C03634=1025.700,9.910,403.538,167.481,46.945,158.663
C03635=1025.707,10.159,403.524,167.485,46.942,158.663
C03636=1025.713,10.408,403.509,167.487,46.939,158.663
C03637=1025.719,10.658,403.495,167.489,46.937,158.663
C03638=1025.725,10.908,403.480,167.492,46.933,158.662
C03639=1025.731,11.192,403.463,167.495,46.930,158.662
C03640=1025.739,11.476,403.446,167.498,46.926,158.662
C03641=1025.745,11.760,403.429,167.501,46.922,158.661
C03642=1025.753,12.044,403.413,167.504,46.919,158.661
C03643=1025.759,12.293,403.398,167.506,46.916,158.661
C03644=1025.765,12.542,403.383,167.510,46.913,158.661
C03645=1025.772,12.792,403.368,167.512,46.910,158.660
C03646=1025.777,13.041,403.354,167.515,46.907,158.660
C03647=1025.784,13.291,403.339,167.517,46.903,158.660
C03648=1025.790,13.540,403.324,167.519,46.900,158.660
C03649=1025.797,13.790,403.309,167.522,46.897,158.659
C03650=1025.802,14.039,403.294,167.525,46.895,158.659
C03651=1025.809,14.289,403.279,167.528,46.892,158.659
C03652=1025.815,14.538,403.264,167.530,46.889,158.659
C03653=1025.821,14.788,403.249,167.532,46.886,158.659
C03654=1025.827,15.037,403.234,167.535,46.883,158.658
C03655=1025.833,15.287,403.219,167.538,46.880,158.658
C03656=1025.839,15.537,403.204,167.541,46.877,158.658
C03657=1025.845,15.785,403.188,167.543,46.874,158.658
C03658=1025.851,16.035,403.173,167.545,46.871,158.657
C03659=1025.857,16.285,403.158,167.548,46.868,158.657
C03660=1025.864,16.534,403.144,167.550,46.865,158.657
C03661=1025.870,16.783,403.129,167.554,46.862,158.657
C03662=1025.875,17.033,403.113,167.556,46.859,158.656
C03663=1025.882,17.283,403.098,167.558,46.856,158.656
C03664=1025.888,17.532,403.083,167.561,46.853,158.656
C03665=1025.895,17.781,403.068,167.563,46.850,158.656
C03666=1025.900,18.031,403.053,167.567,46.847,158.655
C03667=1025.906,18.280,403.038,167.569,46.844,158.655
C03668=1025.912,18.530,403.023,167.571,46.841,158.655
C03669=1025.919,18.780,403.008,167.574,46.838,158.655
C03670=1025.924,19.028,402.992,167.576,46.835,158.655
C03671=1025.931,19.278,402.977,167.580,46.832,158.654
C03672=1025.937,19.528,402.962,167.582,46.829,158.654
C03673=1025.943,19.777,402.947,167.584,46.826,158.654
C03674=1025.949,20.027,402.931,167.587,46.823,158.653
C03675=1025.956,20.276,402.916,167.589,46.820,158.653
C03676=1025.961,20.526,402.901,167.591,46.817,158.653
C03677=1025.967,20.775,402.885,167.595,46.814,158.653
C03678=1025.974,21.024,402.870,167.597,46.811,158.653
C03679=1025.979,21.274,402.855,167.599,46.808,158.652
C03680=1025.986,21.524,402.840,167.602,46.805,158.652
C03681=1025.991,21.773,402.824,167.605,46.803,158.652
C03682=1025.998,22.022,402.809,167.607,46.799,158.652
C03683=1026.004,22.272,402.794,167.610,46.796,158.651
C03684=1026.010,22.521,402.778,167.612,46.793,158.651
C03685=1026.016,22.771,402.763,167.615,46.790,158.651
C03686=1026.023,23.020,402.747,167.617,46.787,158.651
C03687=1026.029,23.270,402.731,167.620,46.785,158.650
C03688=1026.034,23.519,402.717,167.623,46.782,158.650
C03689=1026.040,23.768,402.701,167.625,46.779,158.650
C03690=1026.047,24.018,402.686,167.628,46.775,158.650
C03691=1026.053,24.267,402.671,167.630,46.772,158.649
C03692=1026.059,24.517,402.654,167.632,46.769,158.649
C03693=1026.065,24.766,402.639,167.636,46.766,158.649
C03694=1026.071,25.016,402.623,167.638,46.764,158.649
C03695=1026.078,25.266,402.608,167.640,46.761,158.648
C03696=1026.084,25.514,402.593,167.643,46.758,158.648
C03697=1026.090,25.764,402.577,167.645,46.754,158.648
C03698=1026.096,26.013,402.563,167.648,46.751,158.648
C03699=1026.102,26.263,402.546,167.651,46.748,158.647
C03700=1026.108,26.512,402.531,167.653,46.746,158.647
C03701=1026.114,26.762,402.515,167.656,46.743,158.647
C03702=1026.121,27.011,402.500,167.658,46.740,158.647
C03703=1026.127,27.297,402.482,167.661,46.736,158.646
C03704=1026.135,27.582,402.464,167.664,46.732,158.646
C03705=1026.142,27.867,402.446,167.668,46.729,158.646
C03706=1026.149,28.152,402.429,167.669,46.726,158.645
C03707=1026.154,28.402,402.413,167.673,46.723,158.645
C03708=1026.161,28.651,402.397,167.675,46.720,158.645
C03709=1026.167,28.901,402.382,167.677,46.717,158.645
C03710=1026.173,29.151,402.366,167.680,46.714,158.645
C03711=1026.179,29.400,402.350,167.683,46.711,158.644
C03712=1026.185,29.650,402.334,167.685,46.709,158.644
C03713=1026.191,29.899,402.318,167.688,46.706,158.644
C03714=1026.198,30.148,402.302,167.690,46.703,158.644
C03715=1026.203,30.398,402.287,167.692,46.700,158.643
C03716=1026.210,30.647,402.271,167.695,46.696,158.643
C03717=1026.216,30.896,402.255,167.698,46.693,158.643
C03718=1026.221,31.146,402.239,167.700,46.691,158.643
C03719=1026.228,31.395,402.224,167.703,46.688,158.642
C03720=1026.234,31.645,402.208,167.705,46.685,158.642
C03721=1026.240,31.895,402.192,167.708,46.682,158.642
C03722=1026.246,32.144,402.176,167.711,46.679,158.642
C03723=1026.252,32.393,402.160,167.713,46.676,158.641
C03724=1026.258,32.643,402.145,167.715,46.673,158.641
C03725=1026.265,32.892,402.129,167.718,46.670,158.641
C03726=1026.271,33.141,402.113,167.720,46.667,158.641
C03727=1026.276,33.391,402.097,167.723,46.664,158.640
C03728=1026.283,33.640,402.081,167.726,46.661,158.640
C03729=1026.289,33.890,402.065,167.728,46.658,158.640
C03730=1026.296,34.139,402.049,167.730,46.656,158.640
C03731=1026.301,34.389,402.034,167.734,46.652,158.639
C03732=1026.307,34.638,402.018,167.735,46.649,158.639
C03733=1026.314,34.887,402.002,167.738,46.646,158.639
C03734=1026.320,35.136,401.986,167.741,46.643,158.639
C03735=1026.326,35.386,401.970,167.743,46.640,158.638
C03736=1026.332,35.635,401.955,167.745,46.638,158.638
C03737=1026.338,35.885,401.938,167.749,46.635,158.638
C03738=1026.344,36.134,401.922,167.751,46.631,158.638
C03739=1026.351,36.383,401.906,167.753,46.628,158.637
C03740=1026.356,36.633,401.891,167.756,46.625,158.637
C03741=1026.362,36.883,401.875,167.758,46.623,158.637
C03742=1026.368,37.132,401.858,167.760,46.620,158.637
C03743=1026.375,37.381,401.843,167.764,46.617,158.636
C03744=1026.382,37.631,401.826,167.766,46.614,158.636
C03745=1026.388,37.880,401.810,167.768,46.611,158.636
C03746=1026.394,38.130,401.794,167.770,46.608,158.635
C03747=1026.399,38.379,401.777,167.773,46.605,158.635
C03748=1026.405,38.628,401.761,167.776,46.602,158.635
C03749=1026.411,38.878,401.745,167.778,46.599,158.635
C03750=1026.417,39.127,401.729,167.781,46.596,158.635
C03751=1026.423,39.376,401.712,167.783,46.593,158.634
C03752=1026.430,39.625,401.697,167.785,46.590,158.634
C03753=1026.436,39.875,401.680,167.789,46.587,158.634
C03754=1026.442,40.124,401.664,167.791,46.585,158.634
C03755=1026.448,40.373,401.648,167.793,46.582,158.633
C03756=1026.454,40.624,401.631,167.795,46.579,158.633
C03757=1026.460,40.873,401.615,167.798,46.575,158.633
C03758=1026.466,41.122,401.599,167.801,46.573,158.632
C03759=1026.472,41.372,401.582,167.803,46.570,158.632
C03760=1026.478,41.621,401.566,167.806,46.567,158.632
C03761=1026.484,41.870,401.550,167.808,46.564,158.632
C03762=1026.491,42.119,401.534,167.810,46.561,158.632
C03763=1026.497,42.369,401.518,167.814,46.558,158.631
C03764=1026.503,42.619,401.501,167.816,46.555,158.631
C03765=1026.509,42.868,401.485,167.818,46.553,158.631
C03766=1026.515,43.117,401.469,167.820,46.550,158.631
C03767=1026.522,43.403,401.449,167.823,46.546,158.630
C03768=1026.528,43.688,401.431,167.827,46.543,158.630
C03769=1026.535,43.973,401.412,167.829,46.540,158.630
C03770=1026.542,44.259,401.393,167.832,46.537,158.629
C03771=1026.548,44.508,401.377,167.834,46.534,158.629
C03772=1026.554,44.758,401.360,167.837,46.531,158.629
C03773=1026.560,45.007,401.343,167.839,46.528,158.629
C03774=1026.566,45.256,401.327,167.842,46.525,158.628
C03775=1026.571,45.506,401.310,167.844,46.523,158.628
C03776=1026.578,45.755,401.293,167.847,46.520,158.628
C03777=1026.584,46.004,401.277,167.849,46.517,158.628
C03778=1026.590,46.254,401.260,167.852,46.514,158.628
C03779=1026.596,46.504,401.244,167.854,46.511,158.627
C03780=1026.602,46.753,401.227,167.857,46.508,158.627
C03781=1026.608,47.002,401.210,167.859,46.505,158.627
C03782=1026.614,47.251,401.194,167.862,46.503,158.627
C03783=1026.620,47.501,401.177,167.864,46.500,158.626
C03784=1026.626,47.750,401.160,167.867,46.497,158.626
C03785=1026.632,48.000,401.144,167.869,46.494,158.626
C03786=1026.638,48.249,401.127,167.871,46.491,158.626
C03787=1026.644,48.498,401.110,167.874,46.489,158.625
C03788=1026.650,48.748,401.094,167.877,46.486,158.625
C03789=1026.656,48.997,401.077,167.879,46.482,158.625
C03790=1026.662,49.247,401.061,167.881,46.479,158.624
C03791=1026.668,49.496,401.044,167.883,46.477,158.624
C03792=1026.674,49.745,401.027,167.887,46.474,158.624
C03793=1026.680,49.995,401.011,167.889,46.471,158.624
C03794=1026.687,50.244,400.994,167.891,46.468,158.624
C03795=1026.693,50.493,400.978,167.893,46.465,158.623
C03796=1026.698,50.742,400.960,167.897,46.462,158.623
C03797=1026.705,50.992,400.943,167.899,46.460,158.623
C03798=1026.711,51.241,400.927,167.901,46.457,158.623
C03799=1026.717,51.490,400.910,167.904,46.454,158.622
C03800=1026.723,51.740,400.894,167.906,46.451,158.622
C03801=1026.729,51.990,400.877,167.908,46.448,158.622
C03802=1026.735,52.239,400.860,167.911,46.445,158.621
C03803=1026.741,52.488,400.843,167.914,46.442,158.621
C03804=1026.748,52.737,400.826,167.916,46.439,158.621
C03805=1026.753,52.987,400.809,167.918,46.436,158.621
C03806=1026.759,53.236,400.793,167.922,46.433,158.621
C03807=1026.765,53.485,400.776,167.924,46.430,158.620
C03808=1026.772,53.735,400.759,167.926,46.428,158.620
C03809=1026.778,53.984,400.742,167.928,46.424,158.620
C03810=1026.783,54.234,400.726,167.931,46.421,158.619
C03811=1026.790,54.483,400.708,167.933,46.418,158.619
C03812=1026.796,54.732,400.692,167.936,46.416,158.619
C03813=1026.802,54.981,400.675,167.939,46.413,158.619
C03814=1026.809,55.231,400.658,167.941,46.410,158.618
C03815=1026.814,55.480,400.641,167.943,46.407,158.618
C03816=1026.820,55.730,400.625,167.945,46.404,158.618
C03817=1026.827,55.979,400.607,167.949,46.401,158.618
C03818=1026.833,56.228,400.591,167.951,46.398,158.617
C03819=1026.838,56.477,400.573,167.953,46.395,158.617
C03820=1026.845,56.727,400.557,167.956,46.392,158.617
C03821=1026.851,56.976,400.540,167.958,46.389,158.616
C03822=1026.858,57.226,400.523,167.961,46.386,158.616
C03823=1026.863,57.475,400.506,167.963,46.383,158.616
C03824=1026.869,57.725,400.489,167.966,46.380,158.616
C03825=1026.876,57.974,400.472,167.968,46.377,158.615
C03826=1026.882,58.223,400.456,167.970,46.374,158.615
C03827=1026.888,58.472,400.439,167.973,46.371,158.615
C03828=1026.895,58.722,400.421,167.976,46.368,158.615
C03829=1026.900,58.971,400.405,167.978,46.365,158.614
C03830=1026.907,59.221,400.387,167.981,46.362,158.614
C03831=1026.914,59.506,400.368,167.983,46.359,158.614
C03832=1026.921,59.791,400.349,167.986,46.355,158.613
C03833=1026.928,60.076,400.330,167.989,46.352,158.613
C03834=1026.936,60.361,400.310,167.992,46.349,158.613
C03835=1026.941,60.610,400.293,167.995,46.346,158.613
C03836=1026.948,60.860,400.275,167.997,46.343,158.612
C03837=1026.954,61.109,400.259,168.000,46.340,158.612
C03838=1026.961,61.359,400.242,168.002,46.337,158.612
C03839=1026.966,61.608,400.224,168.004,46.334,158.611
C03840=1026.972,61.857,400.208,168.007,46.330,158.611
C03841=1026.979,62.106,400.191,168.009,46.328,158.611
C03842=1026.985,62.355,400.174,168.012,46.325,158.610
C03843=1026.991,62.605,400.156,168.015,46.322,158.610
C03844=1026.997,62.854,400.139,168.017,46.318,158.610
C03845=1027.004,63.104,400.122,168.019,46.316,158.610
C03846=1027.010,63.353,400.106,168.022,46.313,158.609
C03847=1027.016,63.603,400.088,168.025,46.310,158.609
C03848=1027.023,63.851,400.071,168.027,46.307,158.609
C03849=1027.029,64.101,400.053,168.029,46.304,158.608
C03850=1027.035,64.350,400.036,168.032,46.301,158.608
C03851=1027.041,64.599,400.019,168.034,46.298,158.608
C03852=1027.046,64.849,400.001,168.037,46.295,158.608
C03853=1027.053,65.098,399.984,168.040,46.292,158.608
C03854=1027.059,65.348,399.966,168.042,46.289,158.607
C03855=1027.065,65.596,399.949,168.044,46.287,158.607
C03856=1027.071,65.846,399.931,168.047,46.284,158.607
C03857=1027.077,66.095,399.915,168.049,46.280,158.606
C03858=1027.083,66.345,399.897,168.052,46.278,158.606
C03859=1027.089,66.594,399.880,168.054,46.275,158.606
C03860=1027.096,66.844,399.862,168.056,46.272,158.606
C03861=1027.101,67.093,399.845,168.059,46.269,158.605
C03862=1027.108,67.342,399.827,168.062,46.266,158.605
C03863=1027.113,67.591,399.810,168.064,46.264,158.605
C03864=1027.120,67.841,399.793,168.066,46.261,158.605
C03865=1027.126,68.090,399.775,168.069,46.257,158.604
C03866=1027.132,68.339,399.757,168.071,46.254,158.604
C03867=1027.138,68.588,399.740,168.074,46.252,158.604
C03868=1027.144,68.838,399.722,168.077,46.249,158.604
C03869=1027.150,69.087,399.705,168.079,46.246,158.603
C03870=1027.157,69.336,399.687,168.081,46.243,158.603
C03871=1027.162,69.585,399.670,168.084,46.240,158.603
C03872=1027.168,69.835,399.652,168.086,46.238,158.602
C03873=1027.174,70.084,399.634,168.089,46.235,158.602
C03874=1027.181,70.334,399.617,168.091,46.232,158.602
C03875=1027.187,70.583,399.599,168.094,46.229,158.602
C03876=1027.192,70.832,399.581,168.096,46.226,158.601
C03877=1027.199,71.082,399.564,168.099,46.223,158.601
C03878=1027.205,71.331,399.546,168.101,46.220,158.601
C03879=1027.211,71.581,399.529,168.103,46.217,158.601
C03880=1027.216,71.830,399.511,168.106,46.215,158.600
C03881=1027.223,72.079,399.494,168.109,46.212,158.600
C03882=1027.229,72.328,399.476,168.111,46.209,158.600
C03883=1027.235,72.577,399.457,168.113,46.206,158.600
C03884=1027.241,72.827,399.439,168.117,46.203,158.599
C03885=1027.247,73.076,399.422,168.119,46.200,158.599
C03886=1027.254,73.326,399.405,168.121,46.197,158.599
C03887=1027.259,73.575,399.387,168.123,46.194,158.598
C03888=1027.265,73.824,399.369,168.126,46.191,158.598
C03889=1027.271,74.073,399.351,168.128,46.188,158.598
C03890=1027.278,74.322,399.333,168.131,46.186,158.598
C03891=1027.284,74.572,399.316,168.133,46.183,158.597
C03892=1027.290,74.821,399.298,168.136,46.180,158.597
C03893=1027.296,75.071,399.280,168.138,46.177,158.597
C03894=1027.301,75.320,399.262,168.140,46.174,158.597
C03895=1027.309,75.605,399.242,168.144,46.171,158.596
C03896=1027.316,75.889,399.222,168.147,46.167,158.596
C03897=1027.323,76.175,399.201,168.149,46.164,158.596
C03898=1027.330,76.459,399.181,168.152,46.161,158.595
C03899=1027.336,76.709,399.163,168.154,46.158,158.595
C03900=1027.342,76.958,399.145,168.157,46.155,158.595
C03901=1027.348,77.207,399.127,168.160,46.152,158.595
C03902=1027.354,77.457,399.109,168.162,46.150,158.594
C03903=1027.360,77.706,399.091,168.164,46.147,158.594
C03904=1027.366,77.955,399.073,168.167,46.144,158.594
C03905=1027.372,78.205,399.055,168.170,46.141,158.594
C03906=1027.378,78.454,399.037,168.172,46.138,158.593
C03907=1027.384,78.703,399.019,168.174,46.136,158.593
C03908=1027.390,78.953,399.001,168.177,46.133,158.593
C03909=1027.396,79.202,398.983,168.180,46.130,158.593
C03910=1027.402,79.451,398.965,168.182,46.127,158.592
C03911=1027.408,79.701,398.947,168.184,46.124,158.592
C03912=1027.414,79.949,398.928,168.186,46.121,158.592
C03913=1027.420,80.199,398.910,168.189,46.118,158.591
C03914=1027.426,80.448,398.892,168.192,46.115,158.591
C03915=1027.432,80.697,398.874,168.194,46.113,158.591
C03916=1027.438,80.947,398.856,168.196,46.110,158.591
C03917=1027.444,81.196,398.837,168.199,46.107,158.590
C03918=1027.449,81.445,398.819,168.202,46.104,158.590
C03919=1027.456,81.694,398.801,168.204,46.101,158.590
C03920=1027.462,81.944,398.783,168.206,46.099,158.590
C03921=1027.468,82.192,398.765,168.209,46.096,158.589
C03922=1027.474,82.442,398.747,168.212,46.093,158.589
C03923=1027.480,82.692,398.729,168.214,46.090,158.589
C03924=1027.486,82.940,398.710,168.216,46.088,158.589
C03925=1027.492,83.190,398.692,168.219,46.085,158.588
C03926=1027.498,83.439,398.674,168.222,46.082,158.588
C03927=1027.505,83.689,398.656,168.224,46.079,158.588
C03928=1027.510,83.937,398.638,168.226,46.076,158.587
C03929=1027.517,84.187,398.620,168.229,46.073,158.587
C03930=1027.522,84.436,398.600,168.231,46.070,158.587
C03931=1027.528,84.685,398.583,168.234,46.067,158.587
C03932=1027.534,84.935,398.564,168.236,46.065,158.586
C03933=1027.541,85.184,398.546,168.239,46.062,158.586
C03934=1027.547,85.433,398.528,168.241,46.059,158.586
C03935=1027.553,85.682,398.509,168.244,46.056,158.586
C03936=1027.559,85.932,398.491,168.247,46.053,158.585
C03937=1027.565,86.181,398.473,168.249,46.050,158.585
C03938=1027.571,86.431,398.455,168.251,46.047,158.585
C03939=1027.578,86.680,398.436,168.253,46.044,158.584
C03940=1027.583,86.928,398.418,168.257,46.041,158.584
C03941=1027.590,87.178,398.400,168.259,46.039,158.584
C03942=1027.595,87.427,398.381,168.261,46.036,158.584
C03943=1027.601,87.677,398.363,168.264,46.033,158.584
C03944=1027.608,87.926,398.344,168.267,46.030,158.583
C03945=1027.614,88.175,398.326,168.269,46.027,158.583
C03946=1027.620,88.424,398.308,168.271,46.024,158.583
C03947=1027.626,88.673,398.289,168.274,46.021,158.582
C03948=1027.632,88.923,398.271,168.276,46.018,158.582
C03949=1027.639,89.172,398.253,168.279,46.016,158.582
C03950=1027.645,89.421,398.234,168.282,46.013,158.582
C03951=1027.650,89.671,398.216,168.284,46.010,158.581
C03952=1027.656,89.920,398.197,168.286,46.007,158.581
C03953=1027.663,90.169,398.179,168.289,46.005,158.581
C03954=1027.668,90.418,398.159,168.292,46.002,158.581
C03955=1027.675,90.668,398.141,168.294,45.999,158.580
C03956=1027.680,90.917,398.123,168.296,45.996,158.580
C03957=1027.686,91.166,398.104,168.299,45.993,158.580
C03958=1027.693,91.415,398.085,168.302,45.990,158.580
C03959=1027.699,91.701,398.064,168.304,45.987,158.579
C03960=1027.706,91.985,398.043,168.307,45.984,158.579
C03961=1027.713,92.270,398.021,168.310,45.981,158.579
C03962=1027.719,92.555,398.000,168.312,45.978,158.578
C03963=1027.725,92.804,397.981,168.316,45.975,158.578
C03964=1027.732,93.053,397.963,168.318,45.972,158.578
C03965=1027.737,93.302,397.944,168.320,45.969,158.578
C03966=1027.744,93.551,397.925,168.322,45.967,158.577
C03967=1027.749,93.801,397.906,168.326,45.964,158.577
C03968=1027.756,94.050,397.887,168.328,45.961,158.577
C03969=1027.761,94.299,397.869,168.330,45.958,158.576
C03970=1027.767,94.548,397.850,168.333,45.955,158.576
C03971=1027.774,94.798,397.832,168.335,45.952,158.576
C03972=1027.779,95.047,397.812,168.338,45.949,158.576
C03973=1027.786,95.296,397.794,168.340,45.947,158.575
C03974=1027.792,95.545,397.775,168.343,45.944,158.575
C03975=1027.798,95.795,397.756,168.345,45.941,158.575
C03976=1027.804,96.044,397.737,168.348,45.938,158.575
C03977=1027.810,96.293,397.718,168.350,45.935,158.574
C03978=1027.816,96.542,397.700,168.353,45.932,158.574
C03979=1027.822,96.791,397.681,168.355,45.930,158.574
C03980=1027.828,97.040,397.662,168.358,45.927,158.574
C03981=1027.834,97.289,397.643,168.361,45.924,158.573
C03982=1027.840,97.539,397.624,168.363,45.921,158.573
C03983=1027.846,97.788,397.605,168.365,45.919,158.573
C03984=1027.853,98.037,397.587,168.368,45.915,158.572
C03985=1027.858,98.286,397.567,168.371,45.912,158.572
C03986=1027.865,98.536,397.549,168.373,45.910,158.572
C03987=1027.871,98.785,397.529,168.375,45.907,158.572
C03988=1027.877,99.034,397.511,168.378,45.904,158.571
C03989=1027.883,99.284,397.491,168.381,45.901,158.571
C03990=1027.889,99.533,397.473,168.383,45.899,158.571
C03991=1027.896,99.782,397.454,168.386,45.896,158.571
C03992=1027.901,100.031,397.435,168.388,45.893,158.570
C03993=1027.907,100.281,397.416,168.391,45.890,158.570
C03994=1027.913,100.530,397.397,168.393,45.887,158.570
C03995=1027.918,100.778,397.378,168.396,45.884,158.570
C03996=1027.924,101.028,397.359,168.399,45.882,158.569
C03997=1027.930,101.277,397.340,168.401,45.879,158.569
C03998=1027.937,101.526,397.320,168.403,45.876,158.569
C03999=1027.942,101.775,397.301,168.406,45.873,158.569
C04000=1027.948,102.025,397.282,168.409,45.871,158.568
C04001=1027.954,102.274,397.263,168.411,45.868,158.568
C04002=1027.960,102.523,397.244,168.414,45.865,158.568
C04003=1027.966,102.772,397.224,168.416,45.862,158.568
C04004=1027.972,103.021,397.205,168.419,45.860,158.567
C04005=1027.978,103.271,397.186,168.421,45.857,158.567
C04006=1027.984,103.520,397.167,168.424,45.854,158.567
C04007=1027.990,103.769,397.148,168.426,45.851,158.566
C04008=1027.996,104.018,397.128,168.429,45.849,158.566
C04009=1028.002,104.267,397.109,168.431,45.846,158.566
C04010=1028.008,104.517,397.090,168.434,45.843,158.566
C04011=1028.014,104.766,397.071,168.436,45.840,158.565
C04012=1028.020,105.015,397.051,168.439,45.837,158.565
C04013=1028.026,105.264,397.032,168.442,45.835,158.565
C04014=1028.032,105.513,397.013,168.444,45.832,158.565
C04015=1028.038,105.762,396.993,168.446,45.829,158.564
C04016=1028.044,106.012,396.974,168.450,45.826,158.564
C04017=1028.050,106.261,396.955,168.452,45.823,158.564
C04018=1028.056,106.510,396.936,168.454,45.821,158.564
C04019=1028.062,106.759,396.916,168.457,45.818,158.563
C04020=1028.068,107.008,396.897,168.460,45.815,158.563
C04021=1028.074,107.258,396.878,168.462,45.812,158.563
C04022=1028.080,107.506,396.858,168.464,45.810,158.563
C04023=1028.087,107.791,396.836,168.467,45.806,158.562
C04024=1028.094,108.076,396.814,168.471,45.803,158.562
C04025=1028.101,108.361,396.792,168.474,45.800,158.562
C04026=1028.108,108.646,396.770,168.477,45.797,158.561
C04027=1028.114,108.896,396.750,168.479,45.794,158.561
C04028=1028.120,109.145,396.731,168.481,45.791,158.561
C04029=1028.126,109.394,396.712,168.485,45.788,158.561
C04030=1028.132,109.643,396.692,168.487,45.786,158.560
C04031=1028.138,109.892,396.672,168.489,45.783,158.560
C04032=1028.145,110.141,396.654,168.492,45.780,158.560
C04033=1028.150,110.391,396.634,168.495,45.777,158.560
C04034=1028.156,110.639,396.614,168.497,45.775,158.559
C04035=1028.162,110.889,396.595,168.499,45.772,158.559
C04036=1028.168,111.138,396.575,168.503,45.769,158.559
C04037=1028.174,111.388,396.556,168.505,45.766,158.559
C04038=1028.180,111.637,396.536,168.507,45.764,158.558
C04039=1028.186,111.886,396.516,168.510,45.761,158.558
C04040=1028.192,112.135,396.496,168.513,45.758,158.558
C04041=1028.198,112.384,396.478,168.515,45.755,158.558
C04042=1028.204,112.633,396.458,168.518,45.752,158.557
C04043=1028.210,112.882,396.438,168.520,45.750,158.557
C04044=1028.216,113.131,396.419,168.523,45.747,158.557
C04045=1028.222,113.381,396.398,168.526,45.744,158.557
C04046=1028.228,113.630,396.379,168.528,45.741,158.556
C04047=1028.233,113.879,396.359,168.531,45.739,158.556
C04048=1028.239,114.128,396.339,168.533,45.737,158.556
C04049=1028.245,114.377,396.319,168.536,45.734,158.556
C04050=1028.250,114.626,396.299,168.539,45.731,158.555
C04051=1028.256,114.875,396.279,168.541,45.728,158.555
C04052=1028.262,115.124,396.259,168.543,45.726,158.555
C04053=1028.268,115.373,396.240,168.547,45.723,158.555
C04054=1028.275,115.623,396.219,168.549,45.721,158.554
C04055=1028.281,115.872,396.199,168.551,45.718,158.554
C04056=1028.286,116.122,396.180,168.554,45.715,158.554
C04057=1028.292,116.370,396.160,168.557,45.712,158.554
C04058=1028.298,116.619,396.140,168.559,45.710,158.553
C04059=1028.304,116.868,396.120,168.561,45.707,158.553
C04060=1028.309,117.117,396.100,168.564,45.704,158.553
C04061=1028.316,117.367,396.080,168.567,45.702,158.553
C04062=1028.321,117.616,396.060,168.569,45.699,158.553
C04063=1028.327,117.865,396.040,168.573,45.696,158.552
C04064=1028.333,118.114,396.020,168.575,45.694,158.552
C04065=1028.339,118.363,396.000,168.577,45.691,158.552
C04066=1028.345,118.613,395.980,168.580,45.688,158.552
C04067=1028.351,118.862,395.959,168.583,45.685,158.551
C04068=1028.357,119.111,395.940,168.585,45.683,158.551
C04069=1028.363,119.359,395.920,168.588,45.680,158.551
C04070=1028.368,119.609,395.900,168.591,45.678,158.551
C04071=1028.375,119.858,395.880,168.593,45.675,158.550
C04072=1028.381,120.107,395.860,168.596,45.672,158.550
C04073=1028.386,120.356,395.839,168.598,45.669,158.550
C04074=1028.392,120.605,395.820,168.601,45.667,158.550
C04075=1028.398,120.854,395.800,168.604,45.664,158.549
C04076=1028.405,121.103,395.779,168.606,45.661,158.549
C04077=1028.410,121.353,395.760,168.609,45.658,158.549
C04078=1028.416,121.602,395.739,168.612,45.656,158.549
C04079=1028.422,121.851,395.719,168.614,45.653,158.548
C04080=1028.428,122.100,395.699,168.617,45.651,158.548
C04081=1028.434,122.349,395.679,168.620,45.648,158.548
C04082=1028.440,122.598,395.659,168.622,45.645,158.548
C04083=1028.446,122.848,395.638,168.624,45.643,158.547
C04084=1028.452,123.097,395.618,168.628,45.640,158.547
C04085=1028.458,123.345,395.598,168.630,45.637,158.547
C04086=1028.464,123.594,395.578,168.633,45.634,158.547
C04087=1028.471,123.880,395.555,168.636,45.631,158.546
C04088=1028.478,124.164,395.532,168.639,45.628,158.546
C04089=1028.484,124.449,395.510,168.642,45.625,158.546
C04090=1028.492,124.734,395.487,168.645,45.622,158.546
C04091=1028.497,124.983,395.466,168.647,45.619,158.545
C04092=1028.503,125.232,395.446,168.651,45.616,158.545
C04093=1028.509,125.481,395.426,168.653,45.614,158.545
C04094=1028.516,125.731,395.406,168.656,45.611,158.545
C04095=1028.522,125.979,395.386,168.658,45.608,158.544
C04096=1028.527,126.228,395.365,168.661,45.605,158.544
C04097=1028.534,126.478,395.345,168.664,45.602,158.544
C04098=1028.540,126.726,395.324,168.666,45.600,158.544
C04099=1028.546,126.975,395.304,168.670,45.597,158.543
C04100=1028.552,127.225,395.283,168.672,45.594,158.543
C04101=1028.558,127.474,395.263,168.674,45.591,158.543
C04102=1028.564,127.722,395.243,168.677,45.589,158.543
C04103=1028.571,127.972,395.223,168.680,45.586,158.542
C04104=1028.577,128.221,395.203,168.683,45.583,158.542
C04105=1028.582,128.470,395.183,168.685,45.580,158.542
C04106=1028.588,128.719,395.162,168.687,45.578,158.541
C04107=1028.594,128.968,395.142,168.691,45.575,158.541
C04108=1028.601,129.218,395.122,168.693,45.572,158.541
C04109=1028.606,129.467,395.101,168.696,45.569,158.541
C04110=1028.613,129.715,395.081,168.699,45.566,158.540
C04111=1028.619,129.965,395.060,168.702,45.564,158.540
C04112=1028.625,130.213,395.040,168.704,45.562,158.540
C04113=1028.631,130.463,395.019,168.707,45.559,158.540
C04114=1028.637,130.712,395.000,168.710,45.556,158.540
C04115=1028.642,130.961,394.979,168.712,45.553,158.539
C04116=1028.649,131.210,394.958,168.716,45.550,158.539
C04117=1028.654,131.459,394.937,168.718,45.548,158.539
C04118=1028.661,131.709,394.917,168.720,45.546,158.539
C04119=1028.667,131.957,394.896,168.724,45.543,158.538
C04120=1028.673,132.206,394.876,168.726,45.540,158.538
C04121=1028.678,132.456,394.855,168.729,45.537,158.538
C04122=1028.684,132.704,394.834,168.731,45.535,158.538
C04123=1028.691,132.954,394.813,168.734,45.533,158.538
C04124=1028.696,133.203,394.793,168.737,45.530,158.537
C04125=1028.703,133.452,394.772,168.740,45.527,158.537
C04126=1028.708,133.701,394.751,168.743,45.524,158.537
C04127=1028.714,133.950,394.731,168.745,45.521,158.537
C04128=1028.720,134.199,394.710,168.747,45.519,158.536
C04129=1028.725,134.448,394.689,168.751,45.516,158.536
C04130=1028.732,134.698,394.669,168.753,45.514,158.536
C04131=1028.738,134.946,394.647,168.756,45.511,158.536
C04132=1028.744,135.196,394.627,168.759,45.508,158.535
C04133=1028.750,135.444,394.606,168.761,45.506,158.535
C04134=1028.756,135.694,394.585,168.765,45.503,158.535
C04135=1028.762,135.943,394.565,168.767,45.501,158.535
C04136=1028.767,136.191,394.544,168.770,45.498,158.535
C04137=1028.774,136.441,394.523,168.772,45.495,158.534
C04138=1028.779,136.689,394.502,168.776,45.492,158.534
C04139=1028.786,136.939,394.482,168.778,45.490,158.534
C04140=1028.791,137.187,394.460,168.780,45.488,158.534
C04141=1028.797,137.437,394.440,168.784,45.485,158.533
C04142=1028.804,137.685,394.419,168.786,45.482,158.533
C04143=1028.809,137.935,394.398,168.789,45.479,158.533
C04144=1028.815,138.184,394.377,168.792,45.477,158.533
C04145=1028.822,138.433,394.356,168.795,45.474,158.532
C04146=1028.827,138.682,394.335,168.797,45.471,158.532
C04147=1028.833,138.932,394.314,168.801,45.469,158.532
C04148=1028.839,139.180,394.293,168.803,45.467,158.532
C04149=1028.846,139.429,394.272,168.805,45.464,158.532
C04150=1028.851,139.679,394.251,168.809,45.461,158.531
C04151=1028.857,139.963,394.226,168.812,45.458,158.531
C04152=1028.864,140.247,394.202,168.815,45.455,158.531
C04153=1028.871,140.533,394.179,168.819,45.452,158.531
C04154=1028.878,140.817,394.155,168.821,45.450,158.530
C04155=1028.884,141.066,394.133,168.824,45.447,158.530
C04156=1028.890,141.314,394.112,168.826,45.444,158.530
C04157=1028.895,141.564,394.091,168.830,45.442,158.530
C04158=1028.902,141.812,394.070,168.832,45.439,158.530
C04159=1028.908,142.062,394.049,168.836,45.436,158.529
C04160=1028.913,142.311,394.028,168.838,45.434,158.529
C04161=1028.919,142.560,394.006,168.841,45.431,158.529
C04162=1028.925,142.809,393.985,168.844,45.429,158.529
C04163=1028.931,143.058,393.964,168.847,45.426,158.528
C04164=1028.938,143.307,393.943,168.849,45.423,158.528
C04165=1028.943,143.556,393.922,168.852,45.421,158.528
C04166=1028.949,143.805,393.900,168.855,45.418,158.528
C04167=1028.955,144.055,393.879,168.857,45.416,158.527
C04168=1028.961,144.303,393.858,168.861,45.413,158.527
C04169=1028.967,144.552,393.836,168.863,45.411,158.527
C04170=1028.972,144.801,393.815,168.866,45.408,158.527
C04171=1028.979,145.050,393.795,168.869,45.405,158.527
C04172=1028.985,145.300,393.773,168.872,45.403,158.527
C04173=1028.991,145.548,393.752,168.875,45.400,158.526
C04174=1028.997,145.797,393.730,168.878,45.397,158.526
C04175=1029.003,146.047,393.709,168.880,45.395,158.526
C04176=1029.009,146.295,393.687,168.884,45.393,158.526
C04177=1029.014,146.545,393.666,168.886,45.390,158.525
C04178=1029.020,146.793,393.645,168.889,45.387,158.525
C04179=1029.026,147.043,393.624,168.892,45.385,158.525
C04180=1029.032,147.292,393.602,168.895,45.382,158.525
C04181=1029.038,147.540,393.581,168.897,45.380,158.525
C04182=1029.044,147.789,393.559,168.901,45.377,158.524
C04183=1029.050,148.039,393.537,168.903,45.375,158.524
C04184=1029.056,148.287,393.516,168.907,45.372,158.524
C04185=1029.062,148.536,393.494,168.909,45.370,158.524
C04186=1029.068,148.786,393.473,168.912,45.367,158.524
C04187=1029.074,149.034,393.452,168.915,45.365,158.523
C04188=1029.080,149.283,393.430,168.918,45.362,158.523
C04189=1029.086,149.533,393.408,168.920,45.359,158.523
C04190=1029.092,149.781,393.387,168.924,45.357,158.523
C04191=1029.098,150.030,393.365,168.926,45.354,158.523
C04192=1029.104,150.279,393.344,168.930,45.352,158.522
C04193=1029.109,150.528,393.322,168.932,45.350,158.522
C04194=1029.115,150.777,393.300,168.935,45.347,158.522
C04195=1029.121,151.027,393.279,168.938,45.345,158.522
C04196=1029.127,151.275,393.257,168.941,45.342,158.522
C04197=1029.133,151.524,393.236,168.944,45.339,158.521
C04198=1029.139,151.774,393.214,168.947,45.337,158.521
C04199=1029.145,152.023,393.192,168.949,45.334,158.521
C04200=1029.151,152.271,393.171,168.953,45.332,158.521
C04201=1029.157,152.520,393.149,168.955,45.329,158.521
C04202=1029.163,152.769,393.127,168.958,45.327,158.520
C04203=1029.169,153.019,393.105,168.961,45.325,158.520
C04204=1029.174,153.267,393.084,168.964,45.322,158.520
C04205=1029.180,153.516,393.062,168.967,45.319,158.520
C04206=1029.187,153.766,393.040,168.970,45.317,158.520
C04207=1029.193,154.015,393.019,168.973,45.314,158.519
C04208=1029.198,154.263,392.996,168.976,45.312,158.519
C04209=1029.204,154.512,392.975,168.979,45.309,158.519
C04210=1029.210,154.761,392.953,168.982,45.307,158.519
C04211=1029.216,155.011,392.931,168.985,45.304,158.519
C04212=1029.222,155.259,392.909,168.988,45.302,158.519
C04213=1029.228,155.508,392.887,168.991,45.299,158.518
C04214=1029.234,155.757,392.865,168.993,45.297,158.518
C04215=1029.240,156.041,392.840,168.997,45.295,158.518
C04216=1029.247,156.326,392.816,169.000,45.292,158.518
C04217=1029.254,156.610,392.790,169.003,45.289,158.517
C04218=1029.261,156.894,392.765,169.007,45.286,158.517
C04219=1029.267,157.143,392.743,169.010,45.283,158.517
C04220=1029.273,157.392,392.721,169.013,45.281,158.517
C04221=1029.279,157.641,392.699,169.016,45.278,158.517
C04222=1029.284,157.890,392.677,169.019,45.276,158.517
C04223=1029.290,158.139,392.656,169.022,45.273,158.516
C04224=1029.297,158.387,392.633,169.025,45.271,158.516
C04225=1029.302,158.637,392.611,169.027,45.269,158.516
C04226=1029.308,158.886,392.589,169.031,45.266,158.516
C04227=1029.315,159.135,392.567,169.034,45.263,158.516
C04228=1029.320,159.384,392.545,169.037,45.261,158.515
C04229=1029.326,159.632,392.523,169.040,45.259,158.515
C04230=1029.332,159.882,392.501,169.043,45.257,158.515
C04231=1029.337,160.131,392.478,169.046,45.254,158.515
C04232=1029.344,160.380,392.456,169.049,45.252,158.515
C04233=1029.349,160.629,392.433,169.052,45.250,158.515
C04234=1029.354,160.877,392.411,169.054,45.247,158.514
C04235=1029.361,161.126,392.389,169.058,45.245,158.514
C04236=1029.366,161.375,392.366,169.060,45.243,158.514
C04237=1029.372,161.624,392.344,169.064,45.240,158.514
C04238=1029.377,161.873,392.321,169.067,45.238,158.514
C04239=1029.383,162.122,392.299,169.070,45.236,158.514
C04240=1029.389,162.371,392.277,169.073,45.233,158.513
C04241=1029.394,162.620,392.254,169.076,45.231,158.513
C04242=1029.401,162.869,392.232,169.079,45.229,158.513
C04243=1029.406,163.118,392.209,169.082,45.226,158.513
C04244=1029.412,163.367,392.186,169.085,45.224,158.513
C04245=1029.418,163.616,392.164,169.088,45.222,158.513
C04246=1029.423,163.864,392.142,169.091,45.220,158.513
C04247=1029.429,164.113,392.119,169.093,45.217,158.512
C04248=1029.435,164.362,392.097,169.097,45.215,158.512
C04249=1029.441,164.611,392.074,169.101,45.213,158.512
C04250=1029.447,164.860,392.051,169.103,45.210,158.512
C04251=1029.453,165.109,392.028,169.106,45.208,158.512
C04252=1029.458,165.358,392.006,169.109,45.206,158.512
C04253=1029.464,165.607,391.984,169.112,45.203,158.511
C04254=1029.470,165.856,391.961,169.116,45.201,158.511
C04255=1029.476,166.105,391.938,169.118,45.199,158.511
C04256=1029.481,166.354,391.916,169.122,45.196,158.511
C04257=1029.487,166.602,391.894,169.124,45.194,158.511
C04258=1029.493,166.851,391.871,169.128,45.192,158.511
C04259=1029.499,167.100,391.848,169.131,45.189,158.511
C04260=1029.504,167.349,391.825,169.134,45.187,158.510
C04261=1029.511,167.598,391.803,169.137,45.185,158.510
C04262=1029.516,167.847,391.780,169.140,45.183,158.510
C04263=1029.522,168.096,391.757,169.143,45.180,158.510
C04264=1029.528,168.345,391.734,169.146,45.178,158.510
C04265=1029.534,168.593,391.712,169.149,45.176,158.510
C04266=1029.540,168.842,391.689,169.152,45.173,158.510
C04267=1029.546,169.091,391.666,169.156,45.171,158.509
C04268=1029.551,169.341,391.644,169.158,45.169,158.509
C04269=1029.558,169.589,391.622,169.162,45.166,158.509
C04270=1029.563,169.838,391.599,169.165,45.164,158.509
C04271=1029.573,170.228,391.563,169.169,45.160,158.509
C04272=1029.582,170.617,391.527,169.175,45.157,158.509
C04273=1029.591,171.007,391.491,169.180,45.153,158.508
C04274=1029.600,171.397,391.455,169.184,45.150,158.508
C04275=1029.610,171.789,391.420,169.189,45.146,158.508
C04276=1029.619,172.180,391.384,169.194,45.142,158.508
C04277=1029.629,172.572,391.348,169.200,45.138,158.507
C04278=1029.637,172.965,391.312,169.205,45.134,158.507
C04279=1029.644,173.213,391.290,169.207,45.132,158.507
C04280=1029.650,173.462,391.267,169.211,45.130,158.507
C04281=1029.655,173.711,391.244,169.214,45.127,158.507
C04282=1029.662,173.961,391.220,169.218,45.125,158.507
C04283=1029.668,174.209,391.198,169.220,45.123,158.506
C04284=1029.674,174.458,391.175,169.224,45.121,158.506
C04285=1029.680,174.707,391.151,169.227,45.118,158.506
C04286=1029.686,174.955,391.128,169.230,45.116,158.506
C04287=1029.691,175.204,391.106,169.233,45.114,158.506
C04288=1029.698,175.453,391.083,169.236,45.111,158.506
C04289=1029.704,175.702,391.060,169.240,45.109,158.506
C04290=1029.710,175.951,391.037,169.243,45.107,158.505
C04291=1029.716,176.200,391.014,169.246,45.105,158.505
C04292=1029.722,176.449,390.992,169.249,45.102,158.505
C04293=1029.728,176.697,390.968,169.253,45.100,158.505
C04294=1029.734,176.946,390.945,169.255,45.098,158.505
C04295=1029.740,177.196,390.922,169.259,45.095,158.505
C04296=1029.746,177.445,390.899,169.262,45.093,158.505
C04297=1029.752,177.693,390.876,169.266,45.091,158.504
C04298=1029.758,177.942,390.853,169.268,45.089,158.504
C04299=1029.764,178.190,390.830,169.272,45.086,158.504
C04300=1029.770,178.440,390.806,169.275,45.084,158.504
C04301=1029.776,178.689,390.784,169.279,45.081,158.504
C04302=1029.783,178.937,390.761,169.282,45.079,158.504
C04303=1029.789,179.186,390.738,169.285,45.077,158.504
C04304=1029.795,179.435,390.714,169.288,45.074,158.503
C04305=1029.801,179.684,390.691,169.292,45.072,158.503
C04306=1029.807,179.933,390.668,169.295,45.070,158.503
C04307=1029.813,180.181,390.645,169.299,45.067,158.503
C04308=1029.820,180.431,390.622,169.301,45.065,158.503
C04309=1029.825,180.680,390.599,169.305,45.063,158.503
C04310=1029.831,180.928,390.575,169.308,45.061,158.503
C04311=1029.838,181.177,390.552,169.312,45.058,158.502
C04312=1029.844,181.426,390.530,169.315,45.056,158.502
C04313=1029.850,181.674,390.506,169.319,45.054,158.502
C04314=1029.856,181.923,390.483,169.321,45.052,158.502
C04315=1029.862,182.173,390.460,169.325,45.049,158.502
C04316=1029.868,182.421,390.436,169.328,45.047,158.502
C04317=1029.874,182.670,390.413,169.332,45.045,158.502
C04318=1029.881,182.919,390.390,169.335,45.042,158.502
C04319=1029.886,183.168,390.366,169.339,45.040,158.502
C04320=1029.892,183.416,390.342,169.341,45.038,158.501
C04321=1029.898,183.666,390.319,169.345,45.036,158.501
C04322=1029.904,183.914,390.295,169.348,45.034,158.501
C04323=1029.909,184.163,390.271,169.351,45.032,158.501
C04324=1029.915,184.412,390.248,169.355,45.030,158.501
C04325=1029.922,184.661,390.224,169.358,45.028,158.501
C04326=1029.927,184.909,390.199,169.362,45.026,158.501
C04327=1029.933,185.158,390.176,169.365,45.024,158.501
C04328=1029.938,185.407,390.152,169.368,45.022,158.501
C04329=1029.945,185.656,390.128,169.372,45.020,158.501
C04330=1029.950,185.905,390.105,169.375,45.017,158.501
C04331=1029.956,186.153,390.081,169.379,45.015,158.501
C04332=1029.962,186.402,390.057,169.381,45.013,158.500
C04333=1029.967,186.651,390.033,169.385,45.011,158.500
C04334=1029.973,186.900,390.010,169.388,45.009,158.500
C04335=1029.980,187.149,389.986,169.392,45.007,158.500
C04336=1029.985,187.397,389.961,169.396,45.005,158.500
C04337=1029.991,187.646,389.938,169.398,45.003,158.500
C04338=1029.997,187.896,389.914,169.402,45.001,158.500
C04339=1030.003,188.178,389.887,169.406,44.999,158.500
C04340=1030.011,188.461,389.859,169.410,44.996,158.500
C04341=1030.017,188.746,389.832,169.413,44.994,158.500
C04342=1030.024,189.029,389.805,169.418,44.991,158.500
C04343=1030.030,189.277,389.781,169.420,44.989,158.499
C04344=1030.035,189.526,389.757,169.424,44.987,158.499
C04345=1030.042,189.775,389.733,169.428,44.986,158.499
C04346=1030.047,190.024,389.709,169.431,44.984,158.499
C04347=1030.053,190.273,389.685,169.435,44.981,158.499
C04348=1030.060,190.521,389.662,169.438,44.979,158.499
C04349=1030.065,190.770,389.637,169.442,44.977,158.499
C04350=1030.071,191.019,389.613,169.445,44.975,158.499
C04351=1030.077,191.268,389.589,169.448,44.973,158.499
C04352=1030.083,191.517,389.565,169.452,44.971,158.499
C04353=1030.089,191.765,389.541,169.455,44.969,158.499
C04354=1030.095,192.014,389.517,169.459,44.967,158.499
C04355=1030.101,192.263,389.492,169.463,44.965,158.499
C04356=1030.107,192.512,389.468,169.466,44.963,158.499
C04357=1030.113,192.760,389.445,169.470,44.961,158.498
C04358=1030.119,193.009,389.420,169.472,44.959,158.498
C04359=1030.125,193.258,389.397,169.476,44.957,158.498
C04360=1030.131,193.507,389.372,169.480,44.955,158.498
C04361=1030.137,193.755,389.348,169.483,44.953,158.498
C04362=1030.143,194.004,389.324,169.487,44.951,158.498
C04363=1030.149,194.253,389.300,169.490,44.948,158.498
C04364=1030.155,194.502,389.275,169.494,44.947,158.498
C04365=1030.161,194.750,389.252,169.498,44.945,158.498
C04366=1030.167,195.000,389.227,169.501,44.942,158.498
C04367=1030.173,195.248,389.203,169.505,44.940,158.498
C04368=1030.179,195.497,389.179,169.508,44.938,158.498
C04369=1030.185,195.745,389.154,169.512,44.937,158.498
C04370=1030.192,195.994,389.130,169.516,44.934,158.498
C04371=1030.198,196.243,389.106,169.519,44.932,158.498
C04372=1030.204,196.491,389.082,169.522,44.930,158.497
C04373=1030.210,196.741,389.057,169.525,44.928,158.497
C04374=1030.216,196.989,389.034,169.529,44.927,158.497
C04375=1030.222,197.238,389.009,169.533,44.924,158.497
C04376=1030.229,197.487,388.984,169.536,44.922,158.497
C04377=1030.234,197.735,388.960,169.540,44.920,158.497
C04378=1030.241,197.984,388.936,169.544,44.919,158.497
C04379=1030.246,198.233,388.912,169.547,44.916,158.497
C04380=1030.253,198.481,388.887,169.551,44.914,158.497
C04381=1030.259,198.730,388.863,169.554,44.912,158.497
C04382=1030.265,198.979,388.839,169.558,44.911,158.497
C04383=1030.271,199.228,388.814,169.562,44.908,158.497
C04384=1030.278,199.476,388.789,169.565,44.906,158.497
C04385=1030.283,199.725,388.765,169.569,44.904,158.497
C04386=1030.289,199.974,388.741,169.573,44.903,158.497
C04387=1030.295,200.223,388.717,169.576,44.900,158.497
C04388=1030.302,200.471,388.692,169.580,44.898,158.497
C04389=1030.308,200.720,388.668,169.584,44.897,158.497
C04390=1030.314,200.969,388.642,169.587,44.895,158.497
C04391=1030.320,201.218,388.618,169.591,44.893,158.497
C04392=1030.325,201.466,388.593,169.594,44.891,158.497
C04393=1030.331,201.715,388.568,169.598,44.889,158.496
C04394=1030.338,201.963,388.544,169.602,44.887,158.496
C04395=1030.343,202.212,388.519,169.605,44.885,158.496
C04396=1030.350,202.461,388.494,169.609,44.884,158.496
C04397=1030.356,202.710,388.469,169.613,44.881,158.496
C04398=1030.361,202.958,388.444,169.617,44.880,158.496
C04399=1030.367,203.207,388.419,169.620,44.878,158.496
C04400=1030.374,203.456,388.395,169.624,44.876,158.496
C04401=1030.379,203.704,388.370,169.627,44.874,158.496
C04402=1030.386,203.953,388.345,169.631,44.873,158.496
C04403=1030.411,205.002,388.240,169.988,44.976,158.553
C04404=1030.420,205.367,388.202,169.992,44.974,158.553
C04405=1030.431,205.732,388.163,169.996,44.973,158.553
C04406=1030.441,206.097,388.125,170.000,44.971,158.553
C04407=1030.451,206.462,388.086,170.003,44.970,158.553
C04408=1030.457,206.710,388.060,170.006,44.969,158.553
C04409=1030.465,206.959,388.034,170.009,44.967,158.553
C04410=1030.470,207.207,388.007,170.012,44.967,158.554
C04411=1030.477,207.456,387.981,170.015,44.965,158.554
C04412=1030.484,207.704,387.955,170.018,44.965,158.554
C04413=1030.491,207.953,387.928,170.020,44.964,158.554
C04414=1030.498,208.202,387.902,170.022,44.962,158.554
C04415=1030.504,208.450,387.875,170.025,44.962,158.554
C04416=1030.511,208.699,387.849,170.028,44.960,158.554
C04417=1030.518,208.947,387.823,170.031,44.959,158.554
C04418=1030.525,209.195,387.796,170.034,44.958,158.554
C04419=1030.530,209.444,387.769,170.036,44.957,158.554
C04420=1030.538,209.693,387.743,170.039,44.956,158.554
C04421=1030.545,209.941,387.717,170.042,44.955,158.554
C04422=1030.550,210.190,387.690,170.044,44.954,158.554
C04423=1030.558,210.438,387.664,170.047,44.953,158.554
C04424=1030.564,210.686,387.637,170.050,44.952,158.554
C04425=1030.571,210.935,387.610,170.053,44.951,158.554
C04426=1030.578,211.184,387.583,170.055,44.950,158.554
C04427=1030.584,211.432,387.557,170.058,44.949,158.554
C04428=1030.591,211.681,387.530,170.061,44.948,158.555
C04429=1030.597,211.929,387.504,170.064,44.947,158.555
C04430=1030.604,212.177,387.477,170.067,44.946,158.555
C04431=1030.611,212.426,387.450,170.069,44.945,158.555
C04432=1030.617,212.674,387.423,170.071,44.945,158.555
C04433=1030.624,212.923,387.397,170.074,44.943,158.555
C04434=1030.631,213.172,387.369,170.077,44.943,158.555
C04435=1030.637,213.420,387.343,170.080,44.941,158.555
C04436=1030.644,213.668,387.317,170.083,44.941,158.555
C04437=1030.651,213.917,387.290,170.086,44.939,158.555
C04438=1030.657,214.165,387.263,170.089,44.939,158.555
C04439=1030.664,214.414,387.236,170.092,44.937,158.555
C04440=1030.671,214.663,387.210,170.094,44.937,158.555
C04441=1030.677,214.910,387.182,170.097,44.936,158.555
C04442=1030.684,215.159,387.156,170.100,44.935,158.556
C04443=1030.690,215.408,387.129,170.102,44.934,158.556
C04444=1030.697,215.656,387.102,170.105,44.933,158.556
C04445=1030.704,215.905,387.075,170.108,44.932,158.556
C04446=1030.711,216.154,387.049,170.111,44.931,158.556
C04447=1030.717,216.401,387.021,170.114,44.930,158.556
C04448=1030.724,216.650,386.995,170.117,44.929,158.556
C04449=1030.730,216.899,386.968,170.119,44.928,158.556
C04450=1030.738,217.147,386.941,170.122,44.927,158.556
C04451=1030.744,217.396,386.914,170.125,44.926,158.556
C04452=1030.751,217.644,386.888,170.128,44.925,158.556
C04453=1030.757,217.893,386.860,170.130,44.924,158.556
C04454=1030.764,218.141,386.833,170.134,44.924,158.557
C04455=1030.771,218.389,386.806,170.136,44.922,158.557
C04456=1030.778,218.638,386.780,170.139,44.922,158.557
C04457=1030.784,218.886,386.752,170.142,44.920,158.557
C04458=1030.791,219.135,386.726,170.145,44.920,158.557
C04459=1030.798,219.383,386.698,170.148,44.919,158.557
C04460=1030.807,219.754,386.658,170.152,44.917,158.557
C04461=1030.818,220.125,386.618,170.156,44.917,158.557
C04462=1030.828,220.496,386.577,170.161,44.915,158.557
C04463=1030.837,220.866,386.537,170.165,44.914,158.558
C04464=1030.844,221.115,386.509,170.168,44.913,158.558
C04465=1030.850,221.364,386.482,170.171,44.912,158.558
C04466=1030.857,221.612,386.454,170.174,44.911,158.558
C04467=1030.864,221.860,386.427,170.177,44.910,158.558
C04468=1030.870,222.109,386.400,170.180,44.909,158.558
C04469=1030.877,222.357,386.373,170.182,44.909,158.558
C04470=1030.884,222.606,386.345,170.184,44.908,158.558
C04471=1030.890,222.855,386.318,170.187,44.907,158.558
C04472=1030.897,223.102,386.291,170.190,44.906,158.559
C04473=1030.904,223.351,386.263,170.193,44.905,158.559
C04474=1030.910,223.600,386.236,170.196,44.904,158.559
C04475=1030.917,223.848,386.209,170.199,44.904,158.559
C04476=1030.924,224.096,386.181,170.202,44.902,158.559
C04477=1030.931,224.345,386.154,170.205,44.902,158.559
C04478=1030.937,224.593,386.127,170.208,44.901,158.559
C04479=1030.943,224.841,386.099,170.211,44.900,158.559
C04480=1030.951,225.090,386.072,170.214,44.899,158.559
C04481=1030.957,225.338,386.045,170.217,44.899,158.560
C04482=1030.964,225.587,386.018,170.220,44.898,158.560
C04483=1030.970,225.836,385.990,170.223,44.897,158.560
C04484=1030.977,226.084,385.962,170.226,44.896,158.560
C04485=1030.984,226.332,385.935,170.229,44.895,158.560
C04486=1030.991,226.580,385.908,170.232,44.894,158.560
C04487=1030.997,226.829,385.881,170.235,44.893,158.560
C04488=1031.004,227.077,385.853,170.238,44.893,158.560
C04489=1031.010,227.326,385.825,170.241,44.892,158.560
C04490=1031.018,227.574,385.798,170.244,44.891,158.560
C04491=1031.024,227.822,385.770,170.247,44.890,158.561
C04492=1031.031,228.071,385.742,170.250,44.889,158.561
C04493=1031.038,228.319,385.715,170.252,44.889,158.561
C04494=1031.044,228.568,385.687,170.255,44.888,158.561
C04495=1031.051,228.816,385.659,170.258,44.887,158.561
C04496=1031.057,229.064,385.632,170.261,44.886,158.561
C04497=1031.064,229.312,385.604,170.264,44.886,158.561
C04498=1031.071,229.561,385.576,170.267,44.885,158.562
C04499=1031.077,229.809,385.549,170.270,44.884,158.562
C04500=1031.084,230.058,385.521,170.273,44.884,158.562
C04501=1031.091,230.306,385.493,170.276,44.883,158.562
C04502=1031.097,230.555,385.466,170.279,44.882,158.562
C04503=1031.104,230.803,385.438,170.282,44.881,158.562
C04504=1031.111,231.051,385.410,170.285,44.880,158.562
C04505=1031.117,231.300,385.382,170.288,44.880,158.562
C04506=1031.123,231.549,385.354,170.291,44.879,158.563
C04507=1031.130,231.797,385.326,170.294,44.878,158.563
C04508=1031.137,232.046,385.299,170.297,44.878,158.563
C04509=1031.144,232.293,385.270,170.300,44.877,158.563
C04510=1031.150,232.542,385.242,170.303,44.876,158.563
C04511=1031.157,232.790,385.215,170.306,44.876,158.563
C04512=1031.163,233.039,385.186,170.309,44.875,158.564
C04513=1031.170,233.287,385.159,170.312,44.875,158.564
C04514=1031.177,233.535,385.130,170.315,44.874,158.564
C04515=1031.183,233.784,385.102,170.318,44.873,158.564
C04516=1031.193,234.147,385.062,170.323,44.871,158.564
C04517=1031.202,234.510,385.021,170.327,44.871,158.564
C04518=1031.212,234.873,384.979,170.331,44.870,158.565
C04519=1031.221,235.237,384.939,170.336,44.869,158.565
C04520=1031.228,235.485,384.910,170.339,44.868,158.565
C04521=1031.235,235.733,384.883,170.342,44.867,158.565
C04522=1031.242,235.981,384.855,170.345,44.867,158.565
C04523=1031.249,236.229,384.826,170.348,44.866,158.565
C04524=1031.255,236.478,384.798,170.351,44.865,158.566
C04525=1031.261,236.726,384.770,170.354,44.865,158.566
C04526=1031.268,236.974,384.742,170.357,44.864,158.566
C04527=1031.276,237.223,384.714,170.360,44.863,158.566
C04528=1031.282,237.472,384.686,170.363,44.863,158.566
C04529=1031.288,237.720,384.657,170.366,44.862,158.566
C04530=1031.295,237.968,384.629,170.369,44.861,158.567
C04531=1031.302,238.217,384.602,170.372,44.861,158.567
C04532=1031.309,238.465,384.573,170.375,44.860,158.567
C04533=1031.315,238.713,384.545,170.379,44.859,158.567
C04534=1031.322,238.961,384.516,170.382,44.859,158.567
C04535=1031.328,239.210,384.489,170.385,44.858,158.567
C04536=1031.335,239.457,384.460,170.389,44.858,158.568
C04537=1031.342,239.707,384.432,170.392,44.857,158.568
C04538=1031.349,239.955,384.403,170.395,44.857,158.568
C04539=1031.356,240.203,384.375,170.398,44.856,158.568
C04540=1031.362,240.451,384.346,170.401,44.855,158.568
C04541=1031.369,240.700,384.319,170.404,44.855,158.569
C04542=1031.375,240.948,384.290,170.407,44.854,158.569
C04543=1031.382,241.196,384.262,170.410,44.853,158.569
C04544=1031.388,241.444,384.233,170.413,44.853,158.569
C04545=1031.395,241.693,384.204,170.416,44.853,158.569
C04546=1031.401,241.942,384.176,170.419,44.852,158.569
C04547=1031.408,242.190,384.147,170.423,44.851,158.570
C04548=1031.415,242.438,384.118,170.426,44.851,158.570
C04549=1031.421,242.686,384.090,170.429,44.850,158.570
C04550=1031.427,242.934,384.061,170.432,44.850,158.570
C04551=1031.434,243.182,384.033,170.435,44.849,158.570
C04552=1031.441,243.432,384.004,170.439,44.848,158.571
C04553=1031.448,243.679,383.976,170.442,44.848,158.571
C04554=1031.454,243.928,383.947,170.445,44.847,158.571
C04555=1031.461,244.175,383.918,170.448,44.847,158.571
C04556=1031.467,244.424,383.890,170.451,44.846,158.571
C04557=1031.474,244.673,383.861,170.454,44.846,158.572
C04558=1031.481,244.921,383.832,170.458,44.846,158.572
C04559=1031.487,245.169,383.803,170.461,44.845,158.572
C04560=1031.493,245.417,383.774,170.464,44.844,158.572
C04561=1031.500,245.665,383.745,170.467,44.844,158.572
C04562=1031.507,245.913,383.717,170.470,44.844,158.573
C04563=1031.514,246.162,383.687,170.473,44.843,158.573
C04564=1031.520,246.411,383.659,170.476,44.843,158.573
C04565=1031.526,246.659,383.630,170.480,44.842,158.573
C04566=1031.532,246.907,383.601,170.483,44.842,158.573
C04567=1031.539,247.155,383.572,170.487,44.842,158.574
C04568=1031.546,247.403,383.543,170.490,44.841,158.574
C04569=1031.552,247.652,383.514,170.493,44.840,158.574
C04570=1031.558,247.900,383.485,170.496,44.840,158.574
C04571=1031.565,248.148,383.456,170.499,44.840,158.575
C04572=1031.575,248.505,383.414,170.504,44.839,158.575
C04573=1031.584,248.863,383.372,170.509,44.838,158.575
C04574=1031.593,249.220,383.330,170.513,44.838,158.576
C04575=1031.603,249.576,383.289,170.518,44.837,158.576
C04576=1031.610,249.825,383.259,170.521,44.837,158.576
C04577=1031.616,250.073,383.230,170.524,44.836,158.576
C04578=1031.622,250.321,383.201,170.527,44.836,158.577
C04579=1031.630,250.570,383.172,170.531,44.836,158.577
C04580=1031.636,250.818,383.143,170.535,44.835,158.577
C04581=1031.642,251.066,383.114,170.538,44.835,158.577
C04582=1031.649,251.315,383.085,170.541,44.834,158.577
C04583=1031.656,251.563,383.056,170.544,44.834,158.578
C04584=1031.662,251.811,383.026,170.547,44.833,158.578
C04585=1031.670,252.059,382.997,170.551,44.833,158.578
C04586=1031.676,252.307,382.968,170.555,44.832,158.578
C04587=1031.682,252.555,382.939,170.558,44.832,158.579
C04588=1031.689,252.804,382.910,170.561,44.832,158.579
C04589=1031.696,253.052,382.880,170.564,44.831,158.579
C04590=1031.703,253.300,382.852,170.567,44.831,158.579
C04591=1031.709,253.548,382.822,170.570,44.830,158.580
C04592=1031.716,253.797,382.793,170.575,44.830,158.580
C04593=1031.723,254.045,382.764,170.578,44.829,158.580
C04594=1031.729,254.293,382.734,170.581,44.829,158.580
C04595=1031.735,254.541,382.705,170.584,44.829,158.581
C04596=1031.743,254.790,382.676,170.587,44.829,158.581
C04597=1031.750,255.037,382.646,170.591,44.828,158.581
C04598=1031.756,255.286,382.617,170.594,44.828,158.581
C04599=1031.763,255.534,382.588,170.598,44.827,158.582
C04600=1031.770,255.782,382.558,170.601,44.827,158.582
C04601=1031.777,256.030,382.529,170.604,44.827,158.582
C04602=1031.784,256.279,382.500,170.608,44.826,158.582
C04603=1031.790,256.526,382.470,170.611,44.826,158.583
C04604=1031.797,256.775,382.441,170.614,44.826,158.583
C04605=1031.803,257.023,382.412,170.617,44.825,158.583
C04606=1031.810,257.271,382.382,170.621,44.825,158.583
C04607=1031.817,257.519,382.353,170.625,44.824,158.584
C04608=1031.824,257.767,382.323,170.628,44.824,158.584
C04609=1031.831,258.016,382.294,170.631,44.823,158.584
C04610=1031.838,258.265,382.265,170.634,44.823,158.584
C04611=1031.844,258.512,382.235,170.638,44.822,158.585
C04612=1031.851,258.761,382.205,170.642,44.822,158.585
C04613=1031.858,259.008,382.176,170.645,44.822,158.585
C04614=1031.865,259.257,382.147,170.648,44.822,158.585
C04615=1031.872,259.505,382.117,170.652,44.821,158.586
C04616=1031.879,259.753,382.088,170.655,44.821,158.586
C04617=1031.885,260.001,382.058,170.659,44.821,158.586
C04618=1031.892,260.250,382.029,170.662,44.820,158.586
C04619=1031.899,260.497,381.999,170.666,44.820,158.587
C04620=1031.906,260.746,381.970,170.669,44.819,158.587
C04621=1031.913,260.994,381.940,170.672,44.819,158.587
C04622=1031.920,261.241,381.910,170.677,44.819,158.587
C04623=1031.927,261.490,381.881,170.680,44.818,158.588
C04624=1031.933,261.738,381.850,170.683,44.818,158.588
C04625=1031.940,261.986,381.820,170.686,44.818,158.588
C04626=1031.946,262.234,381.791,170.691,44.818,158.589
C04627=1031.953,262.483,381.761,170.694,44.817,158.589
C04628=1031.963,262.838,381.718,170.698,44.817,158.589
C04629=1031.972,263.194,381.675,170.703,44.817,158.590
C04630=1031.981,263.550,381.632,170.709,44.817,158.590
C04631=1031.991,263.906,381.589,170.713,44.817,158.591
C04632=1031.998,264.154,381.558,170.717,44.816,158.591
C04633=1032.005,264.402,381.529,170.720,44.816,158.591
C04634=1032.012,264.651,381.499,170.724,44.816,158.591
C04635=1032.017,264.898,381.469,170.728,44.815,158.592
C04636=1032.025,265.147,381.439,170.731,44.815,158.592
C04637=1032.032,265.395,381.409,170.735,44.815,158.592
C04638=1032.038,265.642,381.379,170.738,44.815,158.593
C04639=1032.045,265.891,381.348,170.742,44.814,158.593
C04640=1032.052,266.139,381.318,170.745,44.814,158.593
C04641=1032.058,266.387,381.288,170.748,44.814,158.594
C04642=1032.066,266.635,381.258,170.753,44.814,158.594
C04643=1032.072,266.883,381.228,170.756,44.814,158.594
C04644=1032.079,267.131,381.198,170.759,44.814,158.595
C04645=1032.085,267.379,381.167,170.763,44.814,158.595
C04646=1032.092,267.627,381.137,170.767,44.814,158.595
C04647=1032.099,267.875,381.107,170.770,44.813,158.595
C04648=1032.105,268.124,381.076,170.773,44.813,158.596
C04649=1032.112,268.372,381.046,170.777,44.813,158.596
C04650=1032.118,268.620,381.016,170.781,44.813,158.596
C04651=1032.125,268.868,380.986,170.784,44.813,158.597
C04652=1032.132,269.116,380.956,170.788,44.813,158.597
C04653=1032.138,269.363,380.925,170.792,44.813,158.597
C04654=1032.146,269.611,380.895,170.795,44.813,158.598
C04655=1032.152,269.860,380.864,170.799,44.812,158.598
C04656=1032.159,270.108,380.834,170.802,44.812,158.598
C04657=1032.165,270.356,380.803,170.806,44.812,158.599
C04658=1032.172,270.604,380.773,170.810,44.812,158.599
C04659=1032.180,270.852,380.742,170.813,44.812,158.599
C04660=1032.185,271.100,380.712,170.817,44.812,158.600
C04661=1032.192,271.348,380.681,170.821,44.812,158.600
C04662=1032.199,271.596,380.650,170.824,44.812,158.600
C04663=1032.206,271.844,380.620,170.828,44.812,158.601
C04664=1032.213,272.092,380.590,170.832,44.811,158.601
C04665=1032.219,272.340,380.559,170.835,44.812,158.601
C04666=1032.226,272.588,380.528,170.839,44.812,158.602
C04667=1032.233,272.836,380.498,170.843,44.812,158.602
C04668=1032.239,273.084,380.466,170.846,44.812,158.602
C04669=1032.246,273.332,380.437,170.849,44.812,158.603
C04670=1032.252,273.580,380.406,170.854,44.811,158.603
C04671=1032.260,273.828,380.375,170.857,44.811,158.603
C04672=1032.266,274.076,380.344,170.860,44.811,158.604
C04673=1032.273,274.324,380.313,170.865,44.812,158.604
C04674=1032.279,274.572,380.283,170.868,44.812,158.605
C04675=1032.286,274.820,380.252,170.872,44.811,158.605
C04676=1032.293,275.068,380.221,170.876,44.811,158.605
C04677=1032.300,275.316,380.190,170.879,44.811,158.606
C04678=1032.307,275.564,380.159,170.883,44.811,158.606
C04679=1032.313,275.812,380.128,170.887,44.812,158.606
C04680=1032.320,276.061,380.098,170.890,44.812,158.607
C04681=1032.327,276.308,380.067,170.894,44.811,158.607
C04682=1032.333,276.556,380.035,170.898,44.811,158.607
C04683=1032.340,276.804,380.005,170.902,44.811,158.608
C04684=1032.350,277.165,379.960,170.908,44.811,158.608
C04685=1032.360,277.525,379.915,170.913,44.811,158.609
C04686=1032.370,277.885,379.870,170.919,44.812,158.610
C04687=1032.379,278.246,379.825,170.923,44.812,158.610
C04688=1032.386,278.494,379.793,170.928,44.812,158.610
C04689=1032.393,278.742,379.762,170.931,44.812,158.611
C04690=1032.400,278.990,379.731,170.935,44.812,158.611
C04691=1032.407,279.238,379.700,170.939,44.812,158.612
C04692=1032.413,279.486,379.669,170.942,44.813,158.612
C04693=1032.420,279.734,379.638,170.946,44.812,158.612
C04694=1032.427,279.982,379.606,170.950,44.812,158.613
C04695=1032.433,280.230,379.575,170.954,44.813,158.613
C04696=1032.440,280.477,379.544,170.958,44.813,158.614
C04697=1032.446,280.725,379.513,170.962,44.813,158.614
C04698=1032.453,280.973,379.481,170.965,44.813,158.614
C04699=1032.459,281.221,379.450,170.969,44.813,158.615
C04700=1032.466,281.469,379.419,170.973,44.813,158.615
C04701=1032.473,281.717,379.387,170.977,44.813,158.616
C04702=1032.480,281.965,379.356,170.981,44.814,158.616
C04703=1032.487,282.212,379.325,170.984,44.814,158.616
C04704=1032.494,282.460,379.293,170.989,44.814,158.617
C04705=1032.501,282.708,379.262,170.992,44.814,158.617
C04706=1032.507,282.956,379.231,170.997,44.814,158.618
C04707=1032.514,283.204,379.199,171.000,44.814,158.618
C04708=1032.521,283.452,379.168,171.004,44.814,158.618
C04709=1032.528,283.701,379.136,171.008,44.815,158.619
C04710=1032.535,283.949,379.104,171.012,44.814,158.619
C04711=1032.542,284.196,379.073,171.016,44.815,158.620
C04712=1032.548,284.444,379.042,171.020,44.815,158.620
C04713=1032.555,284.692,379.010,171.024,44.815,158.621
C04714=1032.562,284.940,378.979,171.028,44.815,158.621
C04715=1032.568,285.188,378.947,171.031,44.816,158.621
C04716=1032.575,285.436,378.916,171.036,44.815,158.622
C04717=1032.582,285.683,378.884,171.039,44.816,158.622
C04718=1032.589,285.931,378.852,171.043,44.816,158.623
C04719=1032.596,286.180,378.820,171.047,44.816,158.623
C04720=1032.603,286.428,378.789,171.052,44.817,158.624
C04721=1032.610,286.676,378.758,171.055,44.817,158.624
C04722=1032.617,286.923,378.725,171.059,44.817,158.625
C04723=1032.623,287.171,378.694,171.063,44.818,158.625
C04724=1032.630,287.419,378.663,171.067,44.817,158.625
C04725=1032.637,287.667,378.631,171.071,44.818,158.626
C04726=1032.643,287.914,378.598,171.075,44.818,158.626
C04727=1032.650,288.163,378.567,171.079,44.818,158.627
C04728=1032.658,288.410,378.534,171.083,44.819,158.627
C04729=1032.664,288.658,378.503,171.087,44.819,158.628
C04730=1032.671,288.906,378.472,171.091,44.819,158.628
C04731=1032.678,289.153,378.439,171.095,44.820,158.629
C04732=1032.684,289.401,378.407,171.099,44.820,158.629
C04733=1032.692,289.649,378.375,171.102,44.820,158.629
C04734=1032.698,289.897,378.343,171.107,44.820,158.630
C04735=1032.705,290.145,378.312,171.110,44.821,158.630
C04736=1032.711,290.393,378.279,171.115,44.821,158.631
C04737=1032.718,290.641,378.248,171.120,44.822,158.631
C04738=1032.726,290.889,378.215,171.123,44.821,158.632
C04739=1032.733,291.136,378.183,171.127,44.822,158.632
C04740=1032.743,291.509,378.135,171.133,44.823,158.633
C04741=1032.753,291.882,378.087,171.139,44.823,158.634
C04742=1032.763,292.254,378.039,171.146,44.823,158.634
C04743=1032.774,292.626,377.991,171.151,44.824,158.635
C04744=1032.780,292.874,377.958,171.156,44.824,158.636
C04745=1032.788,293.122,377.925,171.159,44.825,158.636
C04746=1032.794,293.370,377.894,171.164,44.825,158.637
C04747=1032.801,293.617,377.861,171.168,44.826,158.637
C04748=1032.808,293.865,377.829,171.172,44.826,158.638
C04749=1032.815,294.113,377.797,171.176,44.826,158.638
C04750=1032.821,294.361,377.765,171.180,44.827,158.639
C04751=1032.829,294.609,377.732,171.184,44.827,158.639
C04752=1032.835,294.857,377.699,171.188,44.828,158.640
C04753=1032.842,295.104,377.667,171.193,44.828,158.640
C04754=1032.848,295.351,377.634,171.197,44.829,158.641
C04755=1032.855,295.600,377.602,171.201,44.829,158.641
C04756=1032.861,295.848,377.569,171.205,44.830,158.642
C04757=1032.868,296.095,377.537,171.209,44.830,158.642
C04758=1032.875,296.344,377.504,171.214,44.831,158.643
C04759=1032.882,296.591,377.471,171.218,44.831,158.643
C04760=1032.889,296.838,377.439,171.222,44.832,158.644
C04761=1032.895,297.086,377.406,171.226,44.832,158.644
C04762=1032.902,297.334,377.373,171.230,44.833,158.645
C04763=1032.908,297.582,377.341,171.234,44.834,158.645
C04764=1032.916,297.829,377.307,171.239,44.834,158.646
C04765=1032.922,298.077,377.275,171.243,44.835,158.646
C04766=1032.929,298.324,377.242,171.247,44.835,158.647
C04767=1032.936,298.572,377.209,171.251,44.836,158.647
C04768=1032.942,298.820,377.177,171.255,44.836,158.648
C04769=1032.949,299.068,377.144,171.260,44.837,158.649
C04770=1032.956,299.316,377.111,171.264,44.837,158.649
C04771=1032.963,299.563,377.079,171.268,44.838,158.650
C04772=1032.970,299.811,377.045,171.273,44.838,158.650
C04773=1032.976,300.058,377.012,171.276,44.839,158.651
C04774=1032.984,300.306,376.979,171.281,44.840,158.651
C04775=1032.990,300.554,376.947,171.286,44.840,158.652
C04776=1032.997,300.802,376.914,171.289,44.841,158.652
C04777=1033.004,301.049,376.880,171.294,44.842,158.653
C04778=1033.011,301.297,376.848,171.298,44.842,158.654
C04779=1033.018,301.545,376.815,171.302,44.843,158.654
C04780=1033.025,301.793,376.781,171.307,44.843,158.655
C04781=1033.031,302.040,376.748,171.311,44.844,158.655
C04782=1033.039,302.288,376.716,171.315,44.844,158.656
C04783=1033.045,302.535,376.682,171.319,44.845,158.656
C04784=1033.052,302.783,376.649,171.324,44.846,158.657
C04785=1033.058,303.031,376.617,171.329,44.846,158.658
C04786=1033.066,303.278,376.583,171.332,44.847,158.658
C04787=1033.073,303.526,376.551,171.337,44.848,158.659
C04788=1033.080,303.774,376.517,171.342,44.848,158.659
C04789=1033.086,304.021,376.484,171.345,44.849,158.660
C04790=1033.094,304.269,376.451,171.350,44.850,158.660
C04791=1033.101,304.517,376.418,171.354,44.850,158.661
C04792=1033.107,304.764,376.385,171.359,44.851,158.662
C04793=1033.115,305.012,376.351,171.363,44.851,158.662
C04794=1033.122,305.260,376.319,171.367,44.852,158.663
C04795=1033.129,305.507,376.285,171.372,44.853,158.663
C04796=1033.140,305.897,376.233,171.379,44.854,158.664
C04797=1033.151,306.286,376.180,171.386,44.855,158.665
C04798=1033.162,306.676,376.128,171.393,44.856,158.666
C04799=1033.173,307.065,376.075,171.400,44.857,158.667
C04800=1033.180,307.313,376.042,171.404,44.858,158.668
C04801=1033.188,307.561,376.009,171.409,44.858,158.668
C04802=1033.195,307.808,375.975,171.413,44.859,158.669
C04803=1033.201,308.056,375.943,171.418,44.860,158.669
C04804=1033.208,308.303,375.909,171.423,44.860,158.670
C04805=1033.216,308.551,375.876,171.427,44.861,158.671
C04806=1033.223,308.799,375.842,171.431,44.862,158.671
C04807=1033.230,309.046,375.809,171.436,44.862,158.672
C04808=1033.237,309.294,375.775,171.440,44.863,158.672
C04809=1033.244,309.541,375.741,171.445,44.864,158.673
C04810=1033.252,309.789,375.709,171.450,44.865,158.674
C04811=1033.259,310.037,375.675,171.455,44.866,158.674
C04812=1033.266,310.284,375.642,171.458,44.866,158.675
C04813=1033.273,310.532,375.608,171.463,44.867,158.676
C04814=1033.280,310.779,375.574,171.468,44.868,158.676
C04815=1033.288,311.027,375.541,171.472,44.868,158.677
C04816=1033.295,311.274,375.507,171.477,44.869,158.677
C04817=1033.302,311.522,375.473,171.482,44.870,158.678
C04818=1033.309,311.769,375.440,171.486,44.871,158.679
C04819=1033.315,312.017,375.405,171.490,44.872,158.679
C04820=1033.323,312.265,375.371,171.495,44.873,158.680
C04821=1033.329,312.513,375.337,171.500,44.874,158.681
C04822=1033.336,312.760,375.303,171.505,44.875,158.681
C04823=1033.343,313.007,375.270,171.509,44.876,158.682
C04824=1033.350,313.255,375.234,171.513,44.877,158.683
C04825=1033.357,313.502,375.201,171.518,44.878,158.683
C04826=1033.364,313.750,375.167,171.523,44.879,158.684
C04827=1033.370,313.998,375.132,171.528,44.880,158.685
C04828=1033.377,314.244,375.098,171.532,44.881,158.686
C04829=1033.384,314.492,375.064,171.537,44.882,158.686
C04830=1033.391,314.740,375.030,171.541,44.883,158.687
C04831=1033.399,314.987,374.995,171.546,44.884,158.688
C04832=1033.405,315.235,374.961,171.551,44.885,158.688
C04833=1033.412,315.483,374.927,171.555,44.886,158.689
C04834=1033.419,315.730,374.892,171.560,44.887,158.690
C04835=1033.426,315.978,374.858,171.565,44.888,158.690
C04836=1033.433,316.226,374.824,171.570,44.889,158.691
C04837=1033.440,316.473,374.789,171.575,44.889,158.692
C04838=1033.447,316.721,374.755,171.578,44.891,158.692
C04839=1033.454,316.968,374.720,171.583,44.892,158.693
C04840=1033.461,317.216,374.686,171.588,44.893,158.694
C04841=1033.468,317.463,374.651,171.593,44.894,158.694
C04842=1033.475,317.711,374.618,171.598,44.894,158.695
C04843=1033.483,317.958,374.583,171.602,44.895,158.696
C04844=1033.489,318.206,374.549,171.607,44.896,158.697
C04845=1033.497,318.453,374.514,171.612,44.898,158.697
C04846=1033.503,318.701,374.480,171.617,44.899,158.698
C04847=1033.511,318.948,374.445,171.622,44.900,158.699
C04848=1033.517,319.196,374.411,171.627,44.901,158.700
C04849=1033.525,319.443,374.376,171.632,44.902,158.700
C04850=1033.532,319.690,374.342,171.636,44.903,158.701
C04851=1033.539,319.938,374.307,171.641,44.904,158.702
C04852=1033.550,320.332,374.251,171.649,44.906,158.703
C04853=1033.562,320.727,374.197,171.656,44.908,158.704
C04854=1033.573,321.121,374.141,171.664,44.909,158.705
C04855=1033.584,321.515,374.086,171.672,44.911,158.706
C04856=1033.592,321.763,374.051,171.677,44.912,158.707
C04857=1033.600,322.010,374.017,171.682,44.913,158.708
C04858=1033.606,322.258,373.982,171.686,44.914,158.709
C04859=1033.614,322.505,373.947,171.692,44.916,158.709
C04860=1033.620,322.753,373.913,171.696,44.917,158.710
C04861=1033.628,323.000,373.878,171.701,44.918,158.711
C04862=1033.635,323.248,373.843,171.706,44.919,158.712
C04863=1033.643,323.495,373.808,171.711,44.920,158.712
C04864=1033.649,323.742,373.773,171.716,44.921,158.713
C04865=1033.658,323.990,373.738,171.721,44.923,158.714
C04866=1033.664,324.237,373.703,171.726,44.924,158.715
C04867=1033.672,324.484,373.668,171.731,44.925,158.716
C04868=1033.679,324.732,373.633,171.736,44.926,158.716
C04869=1033.687,324.979,373.598,171.741,44.927,158.717
C04870=1033.693,325.227,373.563,171.746,44.928,158.718
C04871=1033.702,325.475,373.528,171.751,44.929,158.719
C04872=1033.709,325.722,373.494,171.756,44.931,158.719
C04873=1033.716,325.969,373.459,171.761,44.932,158.720
C04874=1033.724,326.217,373.424,171.766,44.933,158.721
C04875=1033.731,326.464,373.389,171.771,44.934,158.722
C04876=1033.739,326.712,373.354,171.776,44.936,158.723
C04877=1033.746,326.959,373.319,171.781,44.937,158.723
C04878=1033.753,327.206,373.284,171.786,44.938,158.724
C04879=1033.760,327.454,373.249,171.792,44.939,158.725
C04880=1033.768,327.701,373.214,171.797,44.941,158.726
C04881=1033.776,327.949,373.178,171.802,44.942,158.727
C04882=1033.783,328.196,373.143,171.807,44.943,158.727
C04883=1033.791,328.444,373.108,171.812,44.945,158.728
C04884=1033.798,328.691,373.072,171.817,44.946,158.729
C04885=1033.804,328.938,373.037,171.822,44.947,158.730
C04886=1033.812,329.186,373.001,171.827,44.949,158.731
C04887=1033.819,329.433,372.965,171.833,44.950,158.731
C04888=1033.826,329.681,372.930,171.838,44.951,158.732
C04889=1033.833,329.928,372.894,171.843,44.953,158.733
C04890=1033.841,330.176,372.859,171.848,44.954,158.734
C04891=1033.848,330.423,372.823,171.853,44.955,158.735
C04892=1033.856,330.670,372.788,171.858,44.957,158.736
C04893=1033.863,330.917,372.752,171.863,44.959,158.736
C04894=1033.870,331.165,372.716,171.869,44.960,158.737
C04895=1033.877,331.412,372.681,171.874,44.961,158.738
C04896=1033.885,331.659,372.644,171.879,44.963,158.739
C04897=1033.892,331.907,372.609,171.884,44.964,158.740
C04898=1033.899,332.154,372.573,171.889,44.966,158.741
C04899=1033.907,332.401,372.537,171.894,44.967,158.742
C04900=1033.914,332.649,372.502,171.900,44.968,158.742
C04901=1033.922,332.896,372.465,171.905,44.970,158.743
C04902=1033.929,333.143,372.430,171.910,44.971,158.744
C04903=1033.936,333.391,372.394,171.915,44.973,158.745
C04904=1033.943,333.638,372.358,171.920,44.974,158.746
C04905=1033.951,333.885,372.322,171.927,44.976,158.747
C04906=1033.959,334.133,372.286,171.932,44.977,158.748
C04907=1033.966,334.380,372.251,171.937,44.979,158.749
C04908=1033.978,334.770,372.194,171.946,44.981,158.750
C04909=1033.989,335.160,372.137,171.953,44.984,158.752
C04910=1034.000,335.550,372.080,171.962,44.986,158.753
C04911=1034.012,335.939,372.023,171.971,44.989,158.754
C04912=1034.020,336.187,371.987,171.976,44.991,158.755
C04913=1034.027,336.434,371.951,171.981,44.992,158.756
C04914=1034.034,336.682,371.914,171.987,44.994,158.757
C04915=1034.041,336.928,371.878,171.992,44.995,158.758
C04916=1034.049,337.175,371.841,171.997,44.997,158.759
C04917=1034.057,337.423,371.805,172.003,44.999,158.760
C04918=1034.064,337.669,371.769,172.009,45.000,158.761
C04919=1034.071,337.917,371.732,172.014,45.002,158.762
C04920=1034.079,338.165,371.696,172.019,45.003,158.763
C04921=1034.086,338.412,371.660,172.024,45.006,158.764
C04922=1034.094,338.659,371.623,172.030,45.007,158.765
C04923=1034.101,338.906,371.587,172.036,45.009,158.766
C04924=1034.108,339.153,371.550,172.041,45.011,158.767
C04925=1034.116,339.401,371.514,172.047,45.012,158.767
C04926=1034.124,339.648,371.477,172.052,45.014,158.769
C04927=1034.132,339.895,371.441,172.057,45.015,158.769
C04928=1034.139,340.143,371.405,172.064,45.017,158.770
C04929=1034.147,340.390,371.367,172.069,45.019,158.771
C04930=1034.154,340.637,371.331,172.074,45.021,158.772
C04931=1034.161,340.884,371.295,172.080,45.022,158.773
C04932=1034.169,341.131,371.258,172.086,45.024,158.774
C04933=1034.176,341.379,371.221,172.092,45.026,158.775
C04934=1034.184,341.625,371.184,172.097,45.028,158.776
C04935=1034.191,341.873,371.148,172.102,45.030,158.777
C04936=1034.199,342.120,371.111,172.108,45.031,158.778
C04937=1034.206,342.368,371.074,172.114,45.033,158.779
C04938=1034.214,342.614,371.037,172.119,45.035,158.780
C04939=1034.222,342.861,371.000,172.125,45.037,158.781
C04940=1034.229,343.109,370.963,172.130,45.039,158.782
C04941=1034.237,343.356,370.926,172.137,45.041,158.783
C04942=1034.244,343.603,370.889,172.142,45.042,158.784
C04943=1034.252,343.850,370.852,172.147,45.044,158.785
C04944=1034.259,344.098,370.815,172.154,45.046,158.786
C04945=1034.267,344.344,370.778,172.159,45.048,158.787
C04946=1034.274,344.592,370.740,172.165,45.050,158.789
C04947=1034.282,344.839,370.704,172.170,45.052,158.789
C04948=1034.289,345.086,370.667,172.177,45.054,158.790
C04949=1034.297,345.333,370.630,172.182,45.056,158.792
C04950=1034.305,345.580,370.592,172.187,45.058,158.793
C04951=1034.313,345.827,370.555,172.194,45.060,158.794
C04952=1034.320,346.074,370.518,172.199,45.062,158.795
C04953=1034.327,346.321,370.480,172.205,45.064,158.796
C04954=1034.335,346.568,370.443,172.211,45.066,158.797
C04955=1034.343,346.816,370.405,172.217,45.068,158.798
C04956=1034.351,347.063,370.369,172.222,45.070,158.799
C04957=1034.358,347.310,370.331,172.229,45.072,158.800
C04958=1034.366,347.557,370.294,172.234,45.074,158.801
C04959=1034.373,347.804,370.257,172.240,45.076,158.802
C04960=1034.381,348.051,370.220,172.246,45.078,158.803
C04961=1034.389,348.298,370.182,172.252,45.080,158.804
C04962=1034.396,348.546,370.144,172.258,45.082,158.805
C04963=1034.404,348.792,370.107,172.264,45.083,158.806
C04964=1034.417,349.179,370.048,172.273,45.087,158.808
C04965=1034.428,349.566,369.989,172.282,45.090,158.810
C04966=1034.440,349.952,369.930,172.291,45.093,158.812
C04967=1034.453,350.338,369.871,172.301,45.097,158.813
C04968=1034.460,350.585,369.833,172.307,45.099,158.815
C04969=1034.467,350.833,369.796,172.312,45.101,158.816
C04970=1034.476,351.079,369.758,172.319,45.103,158.817
C04971=1034.483,351.327,369.720,172.325,45.105,158.818
C04972=1034.491,351.573,369.682,172.331,45.107,158.819
C04973=1034.498,351.820,369.644,172.337,45.110,158.820
C04974=1034.506,352.068,369.606,172.343,45.112,158.821
C04975=1034.514,352.315,369.568,172.349,45.114,158.823
C04976=1034.522,352.561,369.531,172.356,45.116,158.824
C04977=1034.530,352.809,369.493,172.361,45.118,158.825
C04978=1034.537,353.055,369.455,172.368,45.121,158.826
C04979=1034.545,353.302,369.416,172.373,45.123,158.827
C04980=1034.553,353.550,369.378,172.380,45.125,158.828
C04981=1034.560,353.796,369.340,172.386,45.127,158.829
C04982=1034.569,354.043,369.302,172.392,45.130,158.831
C04983=1034.576,354.290,369.265,172.398,45.132,158.832
C04984=1034.584,354.537,369.226,172.405,45.134,158.833
C04985=1034.592,354.784,369.188,172.410,45.137,158.834
C04986=1034.600,355.031,369.149,172.417,45.139,158.835
C04987=1034.607,355.278,369.112,172.423,45.141,158.837
C04988=1034.616,355.525,369.074,172.430,45.143,158.838
C04989=1034.624,355.772,369.035,172.435,45.145,158.839
C04990=1034.632,356.019,368.997,172.442,45.148,158.840
C04991=1034.640,356.265,368.958,172.448,45.150,158.841
C04992=1034.648,356.513,368.920,172.454,45.153,158.843
C04993=1034.655,356.759,368.882,172.460,45.155,158.844
C04994=1034.663,357.006,368.843,172.467,45.157,158.845
C04995=1034.672,357.253,368.804,172.474,45.160,158.846
C04996=1034.678,357.500,368.766,172.479,45.162,158.848
C04997=1034.687,357.748,368.727,172.486,45.165,158.849
C04998=1034.694,357.994,368.689,172.492,45.167,158.850
C04999=1034.702,358.241,368.650,172.499,45.169,158.851
C05000=1034.711,358.488,368.611,172.504,45.172,158.852
C05001=1034.718,358.734,368.573,172.511,45.174,158.854
C05002=1034.726,358.982,368.534,172.518,45.177,158.855
C05003=1034.735,359.229,368.495,172.524,45.179,158.856
C05004=1034.742,359.475,368.457,172.531,45.181,158.858
C05005=1034.751,359.722,368.418,172.537,45.184,158.859
C05006=1034.759,359.969,368.379,172.543,45.187,158.860
C05007=1034.766,360.216,368.341,172.550,45.189,158.861
C05008=1034.775,360.462,368.302,172.557,45.192,158.863
C05009=1034.783,360.709,368.263,172.563,45.194,158.864
C05010=1034.791,360.956,368.223,172.569,45.197,158.865
C05011=1034.798,361.203,368.185,172.576,45.200,158.867
C05012=1034.807,361.449,368.146,172.582,45.202,158.868
C05013=1034.815,361.697,368.107,172.589,45.204,158.869
C05014=1034.822,361.944,368.067,172.596,45.207,158.871
C05015=1034.831,362.191,368.028,172.602,45.210,158.872
C05016=1034.838,362.437,367.989,172.609,45.212,158.873
C05017=1034.846,362.684,367.949,172.615,45.215,158.874
C05018=1034.854,362.931,367.911,172.622,45.218,158.876
C05019=1034.863,363.177,367.872,172.628,45.221,158.877
C05020=1034.876,363.591,367.805,172.639,45.225,158.879
C05021=1034.890,364.006,367.740,172.651,45.229,158.882
C05022=1034.903,364.419,367.674,172.662,45.234,158.884
C05023=1034.916,364.832,367.607,172.673,45.239,158.886
C05024=1034.924,365.069,367.569,172.680,45.241,158.887
C05025=1034.931,365.305,367.532,172.687,45.244,158.889
C05026=1034.940,365.541,367.494,172.692,45.247,158.890
C05027=1034.948,365.777,367.456,172.699,45.249,158.891
C05028=1034.955,366.014,367.418,172.706,45.252,158.893
C05029=1034.963,366.249,367.380,172.713,45.255,158.894
C05030=1034.971,366.485,367.343,172.719,45.257,158.895
C05031=1034.978,366.722,367.305,172.725,45.260,158.897
C05032=1034.987,366.969,367.265,172.732,45.263,158.898
C05033=1034.996,367.215,367.225,172.739,45.266,158.900
C05034=1035.003,367.461,367.185,172.746,45.269,158.901
C05035=1035.012,367.708,367.146,172.752,45.272,158.903
C05036=1035.019,367.955,367.106,172.760,45.274,158.904
C05037=1035.028,368.202,367.067,172.767,45.277,158.905
C05038=1035.037,368.449,367.027,172.774,45.280,158.907
C05039=1035.045,368.695,366.986,172.781,45.283,158.908
C05040=1035.053,368.942,366.947,172.788,45.286,158.910
C05041=1035.061,369.189,366.907,172.795,45.289,158.911
C05042=1035.070,369.435,366.867,172.802,45.292,158.913
C05043=1035.078,369.681,366.828,172.809,45.295,158.914
C05044=1035.087,369.929,366.788,172.815,45.298,158.916
C05045=1035.095,370.175,366.747,172.822,45.301,158.917
C05046=1035.104,370.421,366.707,172.829,45.304,158.918
C05047=1035.111,370.668,366.667,172.837,45.306,158.920
C05048=1035.119,370.914,366.626,172.844,45.309,158.921
C05049=1035.128,371.162,366.586,172.851,45.312,158.923
C05050=1035.136,371.408,366.546,172.858,45.316,158.924
C05051=1035.144,371.654,366.505,172.865,45.319,158.926
C05052=1035.152,371.901,366.465,172.872,45.322,158.927
C05053=1035.161,372.148,366.424,172.879,45.325,158.929
C05054=1035.170,372.394,366.384,172.887,45.328,158.931
C05055=1035.178,372.640,366.344,172.894,45.331,158.932
C05056=1035.186,372.887,366.303,172.901,45.334,158.933
C05057=1035.194,373.134,366.263,172.908,45.337,158.935
C05058=1035.203,373.380,366.223,172.915,45.340,158.937
C05059=1035.211,373.627,366.182,172.923,45.343,158.938
C05060=1035.219,373.873,366.141,172.930,45.347,158.940
C05061=1035.227,374.120,366.100,172.937,45.350,158.941
C05062=1035.237,374.366,366.060,172.944,45.353,158.943
C05063=1035.245,374.613,366.019,172.952,45.356,158.944
C05064=1035.253,374.860,365.978,172.959,45.359,158.946
C05065=1035.261,375.106,365.938,172.966,45.362,158.947
C05066=1035.270,375.352,365.898,172.975,45.366,158.949
C05067=1035.279,375.599,365.857,172.982,45.369,158.951
C05068=1035.287,375.845,365.816,172.989,45.372,158.952
C05069=1035.296,376.092,365.774,172.996,45.376,158.954
C05070=1035.305,376.338,365.734,173.004,45.379,158.956
C05071=1035.313,376.584,365.693,173.011,45.382,158.957
C05072=1035.322,376.831,365.652,173.018,45.385,158.959
C05073=1035.330,377.078,365.612,173.026,45.389,158.960
C05074=1035.339,377.324,365.571,173.034,45.392,158.962
C05075=1035.347,377.570,365.530,173.042,45.395,158.964
C05076=1035.362,377.984,365.461,173.055,45.401,158.966
C05077=1035.377,378.397,365.392,173.067,45.406,158.969
C05078=1035.391,378.810,365.322,173.080,45.412,158.972
C05079=1035.405,379.224,365.253,173.093,45.418,158.975
C05080=1035.414,379.469,365.212,173.100,45.422,158.976
C05081=1035.422,379.716,365.170,173.108,45.425,158.978
C05082=1035.431,379.963,365.129,173.115,45.428,158.980
C05083=1035.439,380.209,365.087,173.122,45.432,158.981
C05084=1035.448,380.455,365.046,173.131,45.436,158.983
C05085=1035.457,380.701,365.004,173.138,45.439,158.985
C05086=1035.465,380.948,364.962,173.146,45.442,158.987
C05087=1035.474,381.194,364.922,173.154,45.446,158.988
C05088=1035.482,381.440,364.880,173.162,45.450,158.990
C05089=1035.491,381.687,364.838,173.169,45.453,158.992
C05090=1035.500,381.933,364.796,173.177,45.457,158.993
C05091=1035.509,382.180,364.755,173.185,45.461,158.995
C05092=1035.517,382.426,364.713,173.193,45.464,158.997
C05093=1035.526,382.672,364.671,173.202,45.468,158.999
C05094=1035.535,382.918,364.629,173.209,45.471,159.001
C05095=1035.544,383.165,364.588,173.217,45.475,159.002
C05096=1035.553,383.411,364.546,173.225,45.479,159.004
C05097=1035.562,383.657,364.503,173.233,45.482,159.006
C05098=1035.571,383.903,364.462,173.241,45.486,159.008
C05099=1035.580,384.149,364.420,173.249,45.490,159.010
C05100=1035.588,384.396,364.378,173.257,45.493,159.011
C05101=1035.597,384.642,364.336,173.265,45.497,159.013
C05102=1035.606,384.888,364.294,173.273,45.501,159.015
C05103=1035.615,385.135,364.252,173.282,45.505,159.017
C05104=1035.624,385.381,364.210,173.289,45.508,159.018
C05105=1035.633,385.627,364.168,173.297,45.512,159.020
C05106=1035.642,385.873,364.126,173.306,45.516,159.022
C05107=1035.651,386.119,364.083,173.314,45.520,159.024
C05108=1035.660,386.365,364.041,173.322,45.524,159.026
C05109=1035.669,386.611,363.999,173.330,45.527,159.028
C05110=1035.678,386.858,363.957,173.339,45.531,159.030
C05111=1035.688,387.104,363.914,173.346,45.535,159.031
C05112=1035.696,387.350,363.873,173.355,45.538,159.033
C05113=1035.705,387.596,363.830,173.363,45.542,159.035
C05114=1035.714,387.842,363.787,173.372,45.547,159.037
C05115=1035.723,388.089,363.745,173.380,45.550,159.039
C05116=1035.732,388.335,363.702,173.388,45.554,159.041
C05117=1035.741,388.581,363.660,173.397,45.558,159.043
C05118=1035.750,388.827,363.617,173.405,45.562,159.045
C05119=1035.759,389.073,363.574,173.414,45.566,159.047
C05120=1035.768,389.319,363.532,173.422,45.570,159.049
C05121=1035.778,389.565,363.488,173.430,45.574,159.051
C05122=1035.786,389.812,363.447,173.439,45.579,159.053
C05123=1035.795,390.058,363.404,173.447,45.582,159.055
C05124=1035.805,390.304,363.360,173.456,45.586,159.056
C05125=1035.814,390.549,363.318,173.465,45.590,159.058
C05126=1035.823,390.795,363.275,173.473,45.594,159.060
C05127=1035.832,391.042,363.231,173.482,45.599,159.062
C05128=1035.841,391.288,363.189,173.490,45.602,159.064
C05129=1035.850,391.534,363.146,173.499,45.607,159.066
C05130=1035.860,391.780,363.102,173.507,45.611,159.068
C05131=1035.868,392.026,363.059,173.516,45.615,159.070
C05132=1035.877,392.250,363.020,173.524,45.619,159.072
C05133=1035.885,392.474,362.981,173.532,45.623,159.074
C05134=1035.894,392.698,362.941,173.540,45.627,159.076
C05135=1035.903,392.922,362.902,173.548,45.631,159.078
C05136=1035.911,393.146,362.863,173.556,45.634,159.080
C05137=1035.919,393.369,362.824,173.564,45.638,159.082
C05138=1035.928,393.593,362.784,173.572,45.642,159.083
C05139=1035.936,393.817,362.744,173.580,45.646,159.085
C05140=1035.945,394.063,362.700,173.589,45.650,159.087
C05141=1035.955,394.310,362.657,173.597,45.655,159.090
C05142=1035.964,394.555,362.614,173.606,45.659,159.092
C05143=1035.973,394.802,362.570,173.615,45.663,159.094
C05144=1035.983,395.048,362.527,173.625,45.667,159.096
C05145=1035.992,395.293,362.483,173.634,45.672,159.098
C05146=1036.001,395.539,362.439,173.643,45.676,159.100
C05147=1036.010,395.785,362.395,173.651,45.680,159.102
C05148=1036.020,396.031,362.352,173.661,45.685,159.104
C05149=1036.030,396.277,362.308,173.669,45.690,159.106
C05150=1036.039,396.522,362.264,173.678,45.694,159.109
C05151=1036.048,396.769,362.220,173.687,45.699,159.111
C05152=1036.057,397.014,362.176,173.697,45.703,159.113
C05153=1036.068,397.260,362.132,173.706,45.707,159.115
C05154=1036.077,397.506,362.088,173.715,45.712,159.117
C05155=1036.086,397.752,362.044,173.724,45.716,159.119
C05156=1036.095,397.998,362.000,173.734,45.721,159.122
C05157=1036.105,398.244,361.957,173.743,45.726,159.124
C05158=1036.115,398.490,361.912,173.752,45.730,159.126
C05159=1036.125,398.735,361.868,173.761,45.735,159.128
C05160=1036.134,398.982,361.824,173.771,45.739,159.130
C05161=1036.143,399.228,361.779,173.780,45.744,159.133
C05162=1036.154,399.473,361.735,173.789,45.749,159.135
C05163=1036.163,399.719,361.691,173.799,45.753,159.137
C05164=1036.173,399.965,361.646,173.808,45.757,159.139
C05165=1036.182,400.210,361.603,173.817,45.762,159.142
C05166=1036.191,400.456,361.558,173.828,45.767,159.144
C05167=1036.201,400.702,361.513,173.837,45.772,159.146
C05168=1036.211,400.948,361.468,173.846,45.777,159.149
C05169=1036.221,401.193,361.424,173.856,45.781,159.151
C05170=1036.230,401.440,361.379,173.865,45.786,159.153
C05171=1036.240,401.685,361.335,173.875,45.791,159.156
C05172=1036.250,401.931,361.290,173.885,45.796,159.158
C05173=1036.259,402.176,361.245,173.895,45.801,159.160
C05174=1036.269,402.422,361.200,173.904,45.805,159.163
C05175=1036.279,402.668,361.156,173.914,45.810,159.165
C05176=1036.289,402.914,361.111,173.923,45.815,159.167
C05177=1036.299,403.159,361.066,173.934,45.820,159.170
C05178=1036.308,403.405,361.021,173.943,45.825,159.172
C05179=1036.317,403.651,360.976,173.953,45.830,159.175
C05180=1036.327,403.896,360.930,173.962,45.835,159.177
C05181=1036.338,404.142,360.885,173.973,45.840,159.179
C05182=1036.347,404.388,360.840,173.982,45.845,159.182
C05183=1036.356,404.633,360.795,173.992,45.850,159.184
C05184=1036.367,404.879,360.750,174.002,45.855,159.187
C05185=1036.377,405.124,360.704,174.012,45.860,159.189
C05186=1036.386,405.370,360.659,174.022,45.865,159.192
C05187=1036.396,405.616,360.613,174.032,45.870,159.194
C05188=1036.406,405.861,360.568,174.042,45.875,159.197
C05189=1036.416,406.107,360.523,174.053,45.880,159.199
C05190=1036.426,406.352,360.477,174.062,45.886,159.202
C05191=1036.436,406.599,360.431,174.073,45.891,159.204
C05192=1036.446,406.833,360.389,174.082,45.895,159.206
C05193=1036.455,407.066,360.344,174.092,45.900,159.209
C05194=1036.464,407.300,360.301,174.102,45.905,159.211
C05195=1036.475,407.535,360.258,174.112,45.910,159.214
C05196=1036.484,407.769,360.214,174.121,45.915,159.216
C05197=1036.493,408.003,360.171,174.132,45.920,159.219
C05198=1036.504,408.237,360.127,174.141,45.925,159.221
C05199=1036.513,408.471,360.084,174.151,45.930,159.223
C05200=1036.524,408.716,360.038,174.162,45.935,159.226
C05201=1036.533,408.962,359.991,174.173,45.941,159.229
C05202=1036.543,409.207,359.946,174.182,45.946,159.231
C05203=1036.554,409.453,359.900,174.192,45.951,159.234
C05204=1036.565,409.698,359.854,174.203,45.957,159.236
C05205=1036.575,409.944,359.807,174.214,45.962,159.239
C05206=1036.585,410.189,359.762,174.224,45.967,159.242
C05207=1036.595,410.435,359.716,174.235,45.972,159.244
C05208=1036.605,410.681,359.669,174.246,45.978,159.247
C05209=1036.616,410.926,359.623,174.257,45.984,159.250
C05210=1036.626,411.172,359.578,174.267,45.989,159.252
C05211=1036.636,411.418,359.531,174.278,45.994,159.255
C05212=1036.647,411.663,359.484,174.289,46.000,159.258
C05213=1036.657,411.909,359.438,174.299,46.005,159.260
C05214=1036.668,412.154,359.391,174.310,46.011,159.263
C05215=1036.678,412.399,359.345,174.321,46.017,159.266
C05216=1036.688,412.645,359.298,174.332,46.022,159.269
C05217=1036.699,412.890,359.252,174.343,46.027,159.271
C05218=1036.709,413.136,359.204,174.354,46.033,159.274
C05219=1036.720,413.381,359.158,174.365,46.039,159.277
C05220=1036.730,413.627,359.111,174.376,46.045,159.280
C05221=1036.740,413.872,359.064,174.387,46.050,159.283
C05222=1036.751,414.117,359.018,174.398,46.056,159.285
C05223=1036.761,414.362,358.970,174.410,46.062,159.288
C05224=1036.772,414.607,358.924,174.421,46.067,159.291
C05225=1036.783,414.853,358.876,174.432,46.073,159.294
C05226=1036.793,415.099,358.830,174.443,46.079,159.297
C05227=1036.804,415.344,358.783,174.455,46.085,159.300
C05228=1036.814,415.589,358.735,174.465,46.090,159.302
C05229=1036.825,415.835,358.687,174.477,46.096,159.305
C05230=1036.836,416.080,358.641,174.489,46.102,159.308
C05231=1036.846,416.325,358.594,174.500,46.108,159.311
C05232=1036.857,416.570,358.547,174.512,46.114,159.314
C05233=1036.868,416.816,358.499,174.523,46.120,159.317
C05234=1036.878,417.060,358.451,174.535,46.125,159.320
C05235=1036.890,417.306,358.404,174.546,46.132,159.323
C05236=1036.900,417.551,358.357,174.557,46.138,159.326
C05237=1036.911,417.797,358.309,174.569,46.143,159.329
C05238=1036.921,418.042,358.262,174.580,46.149,159.332
C05239=1036.932,418.287,358.213,174.593,46.156,159.335
C05240=1036.944,418.532,358.166,174.604,46.162,159.338
C05241=1036.954,418.778,358.119,174.616,46.168,159.341
C05242=1036.965,419.022,358.071,174.628,46.174,159.344
C05243=1036.976,419.268,358.022,174.639,46.180,159.347
C05244=1036.986,419.513,357.975,174.652,46.186,159.350
C05245=1036.997,419.758,357.927,174.663,46.192,159.353
C05246=1037.008,420.004,357.879,174.675,46.199,159.356
C05247=1037.019,420.248,357.831,174.688,46.205,159.359
C05248=1037.030,420.494,357.782,174.700,46.211,159.363
C05249=1037.041,420.739,357.734,174.712,46.217,159.366
C05250=1037.052,420.984,357.687,174.724,46.223,159.369
C05251=1037.063,421.229,357.638,174.736,46.229,159.372
C05252=1037.074,421.467,357.591,174.748,46.236,159.375
C05253=1037.085,421.706,357.544,174.760,46.242,159.378
C05254=1037.095,421.944,357.497,174.772,46.248,159.381
C05255=1037.107,422.182,357.450,174.783,46.254,159.384
C05256=1037.118,422.421,357.403,174.796,46.260,159.387
C05257=1037.128,422.659,357.355,174.808,46.267,159.391
C05258=1037.139,422.898,357.309,174.820,46.273,159.394
C05259=1037.151,423.136,357.261,174.832,46.279,159.397
C05260=1037.162,423.381,357.213,174.845,46.286,159.400
C05261=1037.173,423.626,357.164,174.857,46.292,159.403
C05262=1037.185,423.871,357.115,174.870,46.298,159.407
C05263=1037.196,424.116,357.067,174.882,46.305,159.410
C05264=1037.207,424.361,357.018,174.895,46.312,159.413
C05265=1037.218,424.606,356.968,174.908,46.318,159.417
C05266=1037.229,424.851,356.919,174.920,46.325,159.420
C05267=1037.241,425.095,356.870,174.933,46.332,159.424
C05268=1037.252,425.340,356.821,174.947,46.338,159.427
C05269=1037.263,425.585,356.772,174.959,46.344,159.430
C05270=1037.275,425.830,356.723,174.972,46.351,159.434
C05271=1037.287,426.075,356.673,174.985,46.358,159.437
C05272=1037.298,426.320,356.624,174.998,46.365,159.440
C05273=1037.309,426.565,356.575,175.012,46.371,159.444
C05274=1037.320,426.810,356.526,175.024,46.378,159.447
C05275=1037.333,427.054,356.476,175.037,46.385,159.451
C05276=1037.344,427.299,356.427,175.050,46.392,159.454
C05277=1037.356,427.545,356.377,175.064,46.398,159.458
C05278=1037.368,427.789,356.328,175.077,46.405,159.461
C05279=1037.378,428.034,356.278,175.091,46.412,159.465
C05280=1037.391,428.279,356.228,175.104,46.419,159.468
C05281=1037.401,428.524,356.178,175.117,46.426,159.472
C05282=1037.414,428.769,356.128,175.131,46.433,159.476
C05283=1037.425,429.013,356.078,175.144,46.440,159.479
C05284=1037.437,429.258,356.028,175.158,46.447,159.483
C05285=1037.448,429.503,355.979,175.171,46.454,159.486
C05286=1037.460,429.748,355.928,175.185,46.461,159.490
C05287=1037.472,429.992,355.878,175.199,46.468,159.494
C05288=1037.484,430.237,355.828,175.213,46.475,159.497
C05289=1037.495,430.482,355.778,175.227,46.482,159.501
C05290=1037.508,430.725,355.727,175.240,46.489,159.505
C05291=1037.519,430.970,355.676,175.254,46.497,159.508
C05292=1037.531,431.215,355.626,175.268,46.504,159.512
C05293=1037.543,431.459,355.577,175.283,46.511,159.516
C05294=1037.555,431.704,355.526,175.296,46.519,159.520
C05295=1037.567,431.949,355.475,175.310,46.525,159.523
C05296=1037.580,432.193,355.425,175.325,46.533,159.527
C05297=1037.591,432.438,355.374,175.339,46.540,159.531
C05298=1037.604,432.683,355.324,175.353,46.547,159.535
C05299=1037.615,432.927,355.272,175.368,46.555,159.539
C05300=1037.627,433.171,355.222,175.382,46.562,159.542
C05301=1037.640,433.416,355.172,175.396,46.569,159.546
C05302=1037.652,433.660,355.120,175.411,46.576,159.550
C05303=1037.665,433.904,355.069,175.425,46.584,159.554
C05304=1037.677,434.150,355.018,175.440,46.591,159.558
C05305=1037.689,434.394,354.967,175.455,46.599,159.562
C05306=1037.701,434.639,354.916,175.469,46.607,159.566
C05307=1037.714,434.883,354.865,175.484,46.614,159.570
C05308=1037.726,435.128,354.814,175.499,46.622,159.574
C05309=1037.738,435.372,354.763,175.513,46.629,159.578
C05310=1037.751,435.617,354.711,175.529,46.637,159.582
C05311=1037.763,435.861,354.659,175.543,46.644,159.586
C05312=1037.775,436.103,354.609,175.558,46.652,159.590
C05313=1037.788,436.344,354.558,175.573,46.660,159.594
C05314=1037.800,436.585,354.507,175.588,46.667,159.598
C05315=1037.813,436.827,354.456,175.603,46.674,159.602
C05316=1037.825,437.068,354.404,175.618,46.682,159.606
C05317=1037.838,437.309,354.353,175.633,46.690,159.610
C05318=1037.850,437.551,354.302,175.649,46.698,159.614
C05319=1037.863,437.792,354.251,175.663,46.706,159.618
C05320=1037.875,438.036,354.199,175.679,46.713,159.622
C05321=1037.887,438.281,354.147,175.694,46.721,159.627
C05322=1037.900,438.525,354.095,175.710,46.729,159.631
C05323=1037.912,438.769,354.043,175.725,46.737,159.635
C05324=1037.925,439.013,353.991,175.741,46.745,159.639
C05325=1037.938,439.258,353.938,175.757,46.753,159.643
C05326=1037.951,439.501,353.886,175.772,46.761,159.648
C05327=1037.964,439.745,353.834,175.789,46.769,159.652
C05328=1037.977,439.990,353.781,175.805,46.777,159.657
C05329=1037.990,440.235,353.729,175.821,46.785,159.661
C05330=1038.003,440.478,353.676,175.836,46.793,159.665
C05331=1038.016,440.722,353.624,175.852,46.801,159.670
C05332=1038.029,440.966,353.571,175.869,46.809,159.674
C05333=1038.042,441.211,353.518,175.885,46.817,159.678
C05334=1038.054,441.454,353.465,175.901,46.826,159.683
C05335=1038.067,441.698,353.412,175.918,46.834,159.687
C05336=1038.081,441.942,353.360,175.934,46.843,159.692
C05337=1038.094,442.186,353.307,175.950,46.851,159.696
C05338=1038.107,442.430,353.254,175.967,46.859,159.701
C05339=1038.120,442.674,353.201,175.983,46.867,159.705
C05340=1038.133,442.918,353.147,176.000,46.875,159.710
C05341=1038.146,443.162,353.094,176.017,46.884,159.714
C05342=1038.160,443.406,353.042,176.034,46.892,159.719
C05343=1038.174,443.650,352.987,176.050,46.901,159.724
C05344=1038.186,443.893,352.934,176.067,46.909,159.728
C05345=1038.200,444.136,352.881,176.085,46.918,159.733
C05346=1038.214,444.380,352.828,176.101,46.926,159.738
C05347=1038.228,444.624,352.775,176.119,46.934,159.742
C05348=1038.242,444.866,352.723,176.136,46.943,159.747
C05349=1038.257,445.110,352.671,176.153,46.951,159.752
C05350=1038.273,445.353,352.619,176.171,46.959,159.756
C05351=1038.289,445.598,352.568,176.187,46.967,159.761
C05352=1038.306,445.841,352.517,176.204,46.975,159.765
C05353=1038.323,446.085,352.467,176.223,46.983,159.770
C05354=1038.340,446.328,352.417,176.240,46.990,159.774
C05355=1038.359,446.572,352.368,176.258,46.998,159.779
C05356=1038.378,446.816,352.319,176.276,47.005,159.784
C05357=1038.397,447.060,352.271,176.293,47.013,159.788
C05358=1038.417,447.305,352.223,176.312,47.020,159.792
C05359=1038.438,447.550,352.175,176.330,47.028,159.797
C05360=1038.460,447.794,352.128,176.347,47.035,159.801
C05361=1038.482,448.038,352.081,176.365,47.042,159.806
C05362=1038.503,448.283,352.035,176.385,47.049,159.810
C05363=1038.526,448.528,351.990,176.403,47.056,159.815
C05364=1038.550,448.773,351.944,176.421,47.063,159.819
C05365=1038.574,449.017,351.900,176.440,47.069,159.824
C05366=1038.598,449.263,351.856,176.458,47.076,159.828
C05367=1038.623,449.508,351.811,176.477,47.082,159.832
C05368=1038.649,449.753,351.768,176.496,47.089,159.837
C05369=1038.675,449.998,351.725,176.515,47.095,159.841
C05370=1038.703,450.243,351.682,176.534,47.101,159.846
C05371=1038.729,450.489,351.641,176.553,47.108,159.850
C05372=1038.774,450.874,351.575,176.582,47.117,159.857
C05373=1038.819,451.258,351.511,176.613,47.126,159.863
C05374=1038.866,451.643,351.448,176.643,47.135,159.870
C05375=1038.914,452.028,351.387,176.673,47.144,159.877
C05376=1038.620,452.080,351.066,176.677,47.217,159.899
C05377=1038.574,451.709,351.125,176.647,47.209,159.893
C05378=1038.528,451.339,351.185,176.618,47.200,159.887
C05379=1038.484,450.968,351.246,176.589,47.192,159.880
C05380=1038.441,450.596,351.309,176.560,47.183,159.874
C05381=1038.413,450.351,351.351,176.541,47.176,159.869
C05382=1038.387,450.105,351.393,176.522,47.170,159.865
C05383=1038.360,449.860,351.436,176.503,47.164,159.861
C05384=1038.334,449.615,351.479,176.484,47.158,159.856
C05385=1038.308,449.370,351.522,176.465,47.152,159.852
C05386=1038.284,449.126,351.567,176.446,47.146,159.848
C05387=1038.259,448.881,351.611,176.428,47.139,159.843
C05388=1038.236,448.635,351.656,176.409,47.132,159.839
C05389=1038.213,448.391,351.702,176.390,47.125,159.834
C05390=1038.190,448.146,351.748,176.372,47.118,159.830
C05391=1038.168,447.901,351.794,176.353,47.112,159.825
C05392=1038.146,447.657,351.841,176.335,47.105,159.821
C05393=1038.125,447.413,351.888,176.318,47.097,159.816
C05394=1038.105,447.168,351.936,176.299,47.090,159.812
C05395=1038.085,446.924,351.984,176.281,47.083,159.807
C05396=1038.065,446.680,352.033,176.264,47.076,159.803
C05397=1038.047,446.435,352.082,176.245,47.068,159.798
C05398=1038.029,446.191,352.131,176.228,47.060,159.794
C05399=1038.012,445.948,352.181,176.211,47.053,159.789
C05400=1037.994,445.705,352.232,176.192,47.045,159.785
C05401=1037.978,445.460,352.282,176.174,47.037,159.780
C05402=1037.962,445.217,352.334,176.157,47.029,159.776
C05403=1037.946,444.973,352.386,176.141,47.021,159.771
C05404=1037.932,444.730,352.437,176.123,47.013,159.766
C05405=1037.917,444.485,352.491,176.105,47.005,159.762
C05406=1037.904,444.241,352.544,176.089,46.996,159.757
C05407=1037.890,443.996,352.598,176.071,46.988,159.752
C05408=1037.877,443.752,352.651,176.054,46.979,159.747
C05409=1037.863,443.508,352.704,176.038,46.971,159.743
C05410=1037.849,443.264,352.757,176.020,46.963,159.738
C05411=1037.836,443.020,352.811,176.004,46.955,159.734
C05412=1037.823,442.776,352.864,175.987,46.946,159.729
C05413=1037.810,442.532,352.918,175.971,46.938,159.725
C05414=1037.797,442.288,352.971,175.954,46.930,159.720
C05415=1037.783,442.044,353.023,175.937,46.922,159.716
C05416=1037.770,441.800,353.076,175.920,46.914,159.711
C05417=1037.757,441.556,353.129,175.904,46.905,159.707
C05418=1037.744,441.312,353.182,175.888,46.897,159.702
C05419=1037.732,441.068,353.234,175.871,46.889,159.698
C05420=1037.718,440.824,353.288,175.855,46.881,159.693
C05421=1037.705,440.581,353.340,175.839,46.873,159.689
C05422=1037.692,440.336,353.393,175.824,46.865,159.685
C05423=1037.679,440.091,353.445,175.807,46.857,159.680
C05424=1037.667,439.848,353.498,175.791,46.849,159.676
C05425=1037.653,439.604,353.550,175.775,46.841,159.671
C05426=1037.640,439.359,353.602,175.759,46.833,159.667
C05427=1037.628,439.115,353.654,175.744,46.825,159.663
C05428=1037.615,438.871,353.707,175.728,46.817,159.659
C05429=1037.602,438.627,353.759,175.712,46.809,159.654
C05430=1037.590,438.383,353.811,175.697,46.802,159.650
C05431=1037.577,438.138,353.863,175.681,46.794,159.646
C05432=1037.564,437.895,353.915,175.665,46.786,159.642
C05433=1037.552,437.653,353.966,175.650,46.778,159.638
C05434=1037.539,437.412,354.017,175.635,46.771,159.634
C05435=1037.527,437.170,354.069,175.619,46.763,159.629
C05436=1037.514,436.929,354.120,175.605,46.755,159.625
C05437=1037.502,436.688,354.171,175.590,46.748,159.621
C05438=1037.489,436.446,354.222,175.574,46.740,159.617
C05439=1037.477,436.205,354.274,175.560,46.733,159.613
C05440=1037.465,435.963,354.324,175.545,46.725,159.609
C05441=1037.453,435.719,354.376,175.530,46.718,159.605
C05442=1037.439,435.474,354.427,175.514,46.710,159.601
C05443=1037.428,435.230,354.479,175.500,46.703,159.597
C05444=1037.416,434.985,354.530,175.485,46.696,159.593
C05445=1037.403,434.741,354.581,175.470,46.688,159.589
C05446=1037.391,434.497,354.632,175.455,46.681,159.585
C05447=1037.379,434.252,354.683,175.440,46.673,159.581
C05448=1037.365,434.007,354.734,175.426,46.666,159.577
C05449=1037.353,433.763,354.786,175.411,46.658,159.574
C05450=1037.341,433.519,354.836,175.397,46.651,159.570
C05451=1037.329,433.274,354.887,175.382,46.644,159.566
C05452=1037.317,433.029,354.938,175.368,46.637,159.562
C05453=1037.304,432.785,354.989,175.354,46.629,159.558
C05454=1037.292,432.540,355.039,175.339,46.622,159.554
C05455=1037.280,432.297,355.090,175.325,46.615,159.551
C05456=1037.268,432.052,355.140,175.310,46.607,159.547
C05457=1037.256,431.807,355.191,175.296,46.601,159.543
